Yaskawa INFORM job: u_tourne2TRJ2.JBI

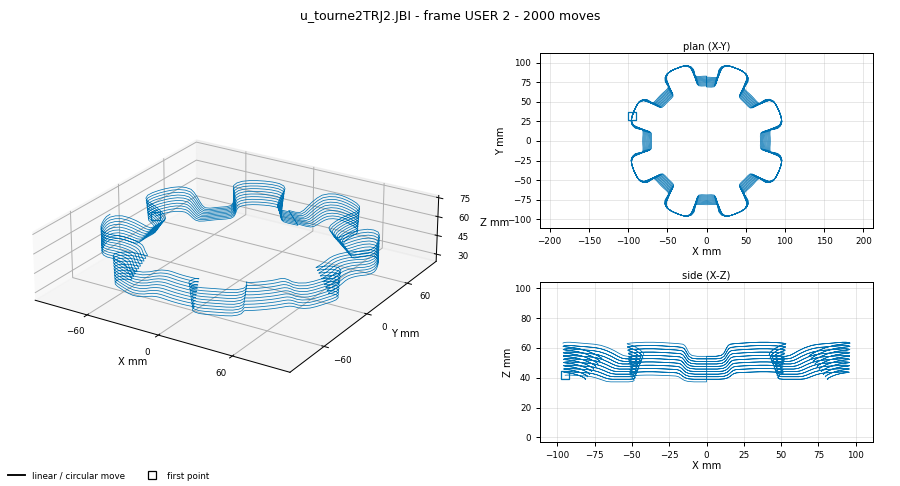
[picture p0: tool path of u_tourne2TRJ2.JBI in frame USER 2, 2000 of 2000 moves have a stored position in this frame; points joined in program order, loops and branches not executed]
/JOB
//NAME u_tourne2TRJ2
///FOLDERNAME DEMO
//POS
///NPOS 2000,0,0,0,0,0
///USER 2
///TOOL 7
///POSTYPE USER
///RECTAN
///RCONF 1,0,0,0,0,0,0,0,0,0,0,0,0,0,0,0,0,0,0,0,0,0,0,0
C00000=-94.679,31.992,41.678,179.9828,-0.0630,0.0000
C00001=-93.214,36.189,41.785,179.9943,-0.0057,0.0000
C00002=-91.502,40.323,41.785,179.9943,-0.0057,0.0000
C00003=-89.570,44.326,41.678,179.9714,-0.0573,0.0000
C00004=-87.153,47.905,41.515,178.9971,-1.0602,0.0000
C00005=-83.964,50.341,41.355,177.9939,-1.0435,0.0000
C00006=-80.606,51.270,41.159,176.0662,-0.0632,0.0000
C00007=-77.545,50.645,40.789,176.2839,1.1369,0.0000
C00008=-74.511,49.565,40.048,179.1806,0.2980,0.0000
C00009=-71.724,48.673,39.090,-174.7314,-1.4558,0.0000
C00010=-69.261,48.447,38.165,-161.9039,-0.3255,0.0000
C00011=-66.868,49.465,37.495,-150.1012,20.4852,0.0000
C00012=-64.059,52.288,37.229,-152.5935,29.6888,0.0000
C00013=-61.349,55.398,37.217,-152.6199,30.0128,0.0000
C00014=-58.451,58.451,37.225,-151.2622,28.7378,0.0000
C00015=-55.398,61.349,37.217,-149.9872,27.3801,0.0000
C00016=-52.288,64.059,37.229,-150.3112,27.4065,0.0000
C00017=-49.465,66.868,37.495,-159.5087,29.8988,0.0000
C00018=-48.447,69.261,38.165,179.6745,18.0961,0.0000
C00019=-48.673,71.724,39.090,178.5442,5.2686,0.0000
C00020=-49.565,74.511,40.048,-179.7020,-0.8194,0.0000
C00021=-50.645,77.545,40.789,-178.8631,-3.7161,0.0000
C00022=-51.270,80.606,41.159,179.9368,-3.9338,0.0000
C00023=-50.341,83.964,41.355,178.9565,-2.0061,0.0000
C00024=-47.905,87.153,41.515,178.9398,-1.0029,0.0000
C00025=-44.326,89.570,41.678,179.9427,-0.0286,0.0000
C00026=-40.323,91.502,41.785,179.9943,-0.0057,0.0000
C00027=-36.189,93.214,41.785,179.9943,-0.0057,0.0000
C00028=-31.992,94.679,41.678,179.9370,-0.0172,0.0000
C00029=-27.752,95.500,41.515,178.5446,-0.0401,0.0000
C00030=-23.775,94.968,41.355,177.8450,0.6823,0.0000
C00031=-20.743,93.250,41.159,177.1708,2.7375,0.0000
C00032=-19.021,90.644,40.789,178.1744,3.4301,0.0000
C00033=-17.640,87.735,40.048,179.6333,0.7850,0.0000
C00034=-16.299,85.134,39.090,-177.2969,-4.7546,0.0000
C00035=-14.718,83.232,38.165,-167.2085,-13.2264,0.0000
C00036=-12.305,82.260,37.495,-146.1467,-8.1019,0.0000
C00037=-8.324,82.270,37.229,-142.4136,2.0895,0.0000
C00038=-4.208,82.553,37.217,-142.2346,2.4206,0.0000
C00039=0.000,82.662,37.225,-142.2064,0.0000,0.0000
C00040=0.000,81.307,38.958,-141.7572,0.0000,0.0000
C00041=4.084,81.202,38.949,-141.7896,-2.4427,0.0000
C00042=8.115,80.931,38.962,-141.9757,-1.8546,0.0000
C00043=12.050,80.963,39.253,-146.2971,9.3078,0.0000
C00044=14.402,82.041,39.987,-169.0733,12.6730,0.0000
C00045=15.932,84.113,41.004,-178.0935,3.7115,0.0000
C00046=17.234,86.943,42.060,179.2949,-1.6619,0.0000
C00047=18.580,90.119,42.880,177.9599,-4.2637,0.0000
C00048=20.259,92.987,43.289,176.7667,-3.4911,0.0000
C00049=23.317,94.913,43.506,177.4435,-0.9062,0.0000
C00050=27.389,95.566,43.684,178.3669,0.0229,0.0000
C00051=31.762,94.755,43.864,179.9255,0.0229,0.0000
C00052=36.110,93.244,43.984,179.9885,0.0057,0.0000
C00053=40.400,91.468,43.984,179.9885,0.0057,0.0000
C00054=44.543,89.461,43.864,179.9312,0.0344,0.0000
C00055=48.209,86.942,43.684,178.8309,1.1405,0.0000
C00056=50.626,83.601,43.506,178.8358,2.4477,0.0000
C00057=51.426,80.077,43.289,-179.8160,4.7437,0.0000
C00058=50.586,76.861,42.880,-178.4251,4.4523,0.0000
C00059=49.291,73.664,42.060,-179.3236,1.6734,0.0000
C00060=48.211,70.742,41.004,178.7192,-3.9688,0.0000
C00061=47.828,68.195,39.987,178.7094,-16.4610,0.0000
C00062=48.729,65.770,39.253,-160.4136,-30.4355,0.0000
C00063=51.488,62.965,38.962,-150.0635,-27.9250,0.0000
C00064=54.531,60.307,38.949,-149.5964,-27.7691,0.0000
C00065=57.493,57.493,38.958,-150.8693,-29.1307,0.0000
C00066=60.306,54.531,38.949,-152.2309,-30.4036,0.0000
C00067=62.965,51.488,38.962,-152.0750,-29.9365,0.0000
C00068=65.770,48.729,39.253,-149.5645,-19.5864,0.0000
C00069=68.195,47.828,39.987,-163.5390,1.2906,0.0000
C00070=70.742,48.211,41.004,-176.0312,1.2808,0.0000
C00071=73.664,49.291,42.060,178.3266,-0.6764,0.0000
C00072=76.861,50.586,42.880,175.5477,-1.5749,0.0000
C00073=80.077,51.426,43.289,175.2563,-0.1840,0.0000
C00074=83.601,50.626,43.506,177.5523,1.1642,0.0000
C00075=86.942,48.209,43.684,178.8595,1.1691,0.0000
C00076=89.461,44.543,43.864,179.9656,0.0688,0.0000
C00077=91.468,40.400,43.984,179.9943,0.0115,0.0000
C00078=93.244,36.110,43.984,179.9943,0.0115,0.0000
C00079=94.755,31.762,43.864,179.9771,0.0745,0.0000
C00080=95.566,27.389,43.684,179.9771,1.6331,0.0000
C00081=94.913,23.317,43.506,-179.0938,2.5565,0.0000
C00082=92.987,20.259,43.289,-176.5089,3.2333,0.0000
C00083=90.119,18.580,42.880,-175.7363,2.0401,0.0000
C00084=86.943,17.234,42.060,-178.3381,0.7051,0.0000
C00085=84.113,15.932,41.004,176.2885,-1.9065,0.0000
C00086=82.041,14.402,39.987,167.3270,-10.9267,0.0000
C00087=80.963,12.050,39.253,170.6922,-33.7029,0.0000
C00088=80.931,8.115,38.962,-178.1454,-38.0243,0.0000
C00089=81.202,4.084,38.949,-177.5573,-38.2104,0.0000
C00090=81.307,0.000,38.958,180.0000,-38.2428,0.0000
C00091=81.202,-4.084,38.949,177.5573,-38.2104,0.0000
C00092=80.931,-8.116,38.962,178.1454,-38.0243,0.0000
C00093=80.963,-12.050,39.253,-170.6922,-33.7029,0.0000
C00094=82.041,-14.402,39.987,-167.3270,-10.9267,0.0000
C00095=84.113,-15.932,41.004,-176.2885,-1.9065,0.0000
C00096=86.943,-17.234,42.060,178.3381,0.7051,0.0000
C00097=90.119,-18.580,42.880,175.7363,2.0401,0.0000
C00098=92.987,-20.259,43.289,176.5089,3.2333,0.0000
C00099=94.913,-23.317,43.506,179.0938,2.5565,0.0000
C00100=95.566,-27.389,43.684,-179.9771,1.6331,0.0000
C00101=94.755,-31.762,43.864,-179.9771,0.0745,0.0000
C00102=93.244,-36.110,43.984,-179.9943,0.0115,0.0000
C00103=91.468,-40.400,43.984,-179.9943,0.0115,0.0000
C00104=89.461,-44.543,43.864,-179.9656,0.0688,0.0000
C00105=86.942,-48.209,43.684,-178.8595,1.1691,0.0000
C00106=83.601,-50.626,43.506,-177.5523,1.1642,0.0000
C00107=80.077,-51.426,43.289,-175.2563,-0.1840,0.0000
C00108=76.861,-50.586,42.880,-175.5477,-1.5749,0.0000
C00109=73.664,-49.291,42.060,-178.3266,-0.6764,0.0000
C00110=70.742,-48.211,41.004,176.0312,1.2808,0.0000
C00111=68.195,-47.828,39.987,163.5390,1.2906,0.0000
C00112=65.770,-48.729,39.253,149.5645,-19.5864,0.0000
C00113=62.965,-51.488,38.962,152.0750,-29.9365,0.0000
C00114=60.307,-54.531,38.949,152.2309,-30.4036,0.0000
C00115=57.493,-57.493,38.958,150.8693,-29.1307,0.0000
C00116=54.531,-60.306,38.949,149.5964,-27.7691,0.0000
C00117=51.488,-62.965,38.962,150.0635,-27.9250,0.0000
C00118=48.729,-65.770,39.253,160.4136,-30.4355,0.0000
C00119=47.828,-68.195,39.987,-178.7094,-16.4610,0.0000
C00120=48.211,-70.742,41.004,-178.7192,-3.9688,0.0000
C00121=49.291,-73.664,42.060,179.3236,1.6734,0.0000
C00122=50.586,-76.861,42.880,178.4251,4.4523,0.0000
C00123=51.426,-80.077,43.289,179.8160,4.7437,0.0000
C00124=50.626,-83.601,43.506,-178.8358,2.4477,0.0000
C00125=48.209,-86.942,43.684,-178.8309,1.1405,0.0000
C00126=44.543,-89.461,43.864,-179.9312,0.0344,0.0000
C00127=40.400,-91.468,43.984,-179.9885,0.0057,0.0000
C00128=36.110,-93.244,43.984,-179.9885,0.0057,0.0000
C00129=31.762,-94.755,43.864,-179.9255,0.0229,0.0000
C00130=27.389,-95.566,43.684,-178.3669,0.0229,0.0000
C00131=23.317,-94.913,43.506,-177.4435,-0.9062,0.0000
C00132=20.259,-92.987,43.289,-176.7667,-3.4911,0.0000
C00133=18.580,-90.119,42.880,-177.9599,-4.2637,0.0000
C00134=17.234,-86.943,42.060,-179.2949,-1.6619,0.0000
C00135=15.932,-84.113,41.004,178.0935,3.7115,0.0000
C00136=14.402,-82.041,39.987,169.0733,12.6730,0.0000
C00137=12.050,-80.963,39.253,146.2971,9.3078,0.0000
C00138=8.115,-80.931,38.962,141.9757,-1.8546,0.0000
C00139=4.084,-81.202,38.949,141.7896,-2.4427,0.0000
C00140=0.000,-81.307,38.958,141.7572,0.0000,0.0000
C00141=0.000,-81.307,38.958,141.7572,0.0000,0.0000
C00142=-4.084,-81.202,38.949,141.7896,2.4427,0.0000
C00143=-8.116,-80.931,38.962,141.9757,1.8546,0.0000
C00144=-12.050,-80.963,39.253,146.2971,-9.3078,0.0000
C00145=-14.402,-82.041,39.987,169.0733,-12.6730,0.0000
C00146=-15.932,-84.113,41.004,178.0935,-3.7115,0.0000
C00147=-17.234,-86.943,42.060,-179.2949,1.6619,0.0000
C00148=-18.580,-90.119,42.880,-177.9599,4.2637,0.0000
C00149=-20.259,-92.987,43.289,-176.7667,3.4911,0.0000
C00150=-23.317,-94.913,43.506,-177.4435,0.9062,0.0000
C00151=-27.389,-95.566,43.684,-178.3669,-0.0229,0.0000
C00152=-31.762,-94.755,43.864,-179.9255,-0.0229,0.0000
C00153=-36.110,-93.244,43.984,-179.9885,-0.0057,0.0000
C00154=-40.400,-91.468,43.984,-179.9885,-0.0057,0.0000
C00155=-44.543,-89.461,43.864,-179.9312,-0.0344,0.0000
C00156=-48.209,-86.942,43.684,-178.8309,-1.1405,0.0000
C00157=-50.626,-83.601,43.506,-178.8358,-2.4477,0.0000
C00158=-51.426,-80.077,43.289,179.8160,-4.7437,0.0000
C00159=-50.586,-76.861,42.880,178.4251,-4.4523,0.0000
C00160=-49.291,-73.664,42.060,179.3236,-1.6734,0.0000
C00161=-48.211,-70.742,41.004,-178.7192,3.9688,0.0000
C00162=-47.828,-68.195,39.987,-178.7094,16.4610,0.0000
C00163=-48.729,-65.770,39.253,160.4136,30.4355,0.0000
C00164=-51.488,-62.965,38.962,150.0635,27.9250,0.0000
C00165=-54.531,-60.307,38.949,149.5964,27.7691,0.0000
C00166=-57.493,-57.493,38.958,150.8693,29.1307,0.0000
C00167=-60.306,-54.531,38.949,152.2309,30.4036,0.0000
C00168=-62.965,-51.488,38.962,152.0750,29.9365,0.0000
C00169=-65.770,-48.729,39.253,149.5645,19.5864,0.0000
C00170=-68.195,-47.828,39.987,163.5390,-1.2906,0.0000
C00171=-70.742,-48.211,41.004,176.0312,-1.2808,0.0000
C00172=-73.664,-49.291,42.060,-178.3266,0.6764,0.0000
C00173=-76.861,-50.586,42.880,-175.5477,1.5749,0.0000
C00174=-80.077,-51.426,43.289,-175.2563,0.1840,0.0000
C00175=-83.601,-50.626,43.506,-177.5523,-1.1642,0.0000
C00176=-86.942,-48.209,43.684,-178.8595,-1.1691,0.0000
C00177=-89.461,-44.543,43.864,-179.9656,-0.0688,0.0000
C00178=-91.468,-40.400,43.984,-179.9943,-0.0115,0.0000
C00179=-93.244,-36.110,43.984,-179.9943,-0.0115,0.0000
C00180=-94.755,-31.762,43.864,-179.9771,-0.0745,0.0000
C00181=-95.566,-27.389,43.684,-179.9771,-1.6331,0.0000
C00182=-94.913,-23.317,43.506,179.0938,-2.5565,0.0000
C00183=-92.987,-20.259,43.289,176.5089,-3.2333,0.0000
C00184=-90.119,-18.580,42.880,175.7363,-2.0401,0.0000
C00185=-86.943,-17.234,42.060,178.3381,-0.7051,0.0000
C00186=-84.113,-15.932,41.004,-176.2885,1.9065,0.0000
C00187=-82.041,-14.402,39.987,-167.3270,10.9267,0.0000
C00188=-80.963,-12.050,39.253,-170.6922,33.7029,0.0000
C00189=-80.931,-8.115,38.962,178.1454,38.0243,0.0000
C00190=-81.202,-4.084,38.949,177.5573,38.2104,0.0000
C00191=-81.307,0.000,38.958,-180.0000,38.2428,0.0000
C00192=-81.202,4.084,38.949,-177.5573,38.2104,0.0000
C00193=-80.931,8.116,38.962,-178.1454,38.0243,0.0000
C00194=-80.963,12.050,39.253,170.6922,33.7029,0.0000
C00195=-82.041,14.402,39.987,167.3270,10.9267,0.0000
C00196=-84.113,15.932,41.004,176.2885,1.9065,0.0000
C00197=-86.943,17.234,42.060,-178.3381,-0.7051,0.0000
C00198=-90.119,18.580,42.880,-175.7363,-2.0401,0.0000
C00199=-92.987,20.259,43.289,-176.5089,-3.2333,0.0000
C00200=-94.913,23.317,43.506,-179.0938,-2.5565,0.0000
C00201=-95.566,27.389,43.684,179.9771,-1.6331,0.0000
C00202=-94.755,31.762,43.864,179.9771,-0.0745,0.0000
C00203=-93.244,36.110,43.984,179.9943,-0.0115,0.0000
C00204=-91.468,40.400,43.984,179.9943,-0.0115,0.0000
C00205=-89.461,44.543,43.864,179.9656,-0.0688,0.0000
C00206=-86.942,48.209,43.684,178.8595,-1.1691,0.0000
C00207=-83.601,50.626,43.506,177.5523,-1.1642,0.0000
C00208=-80.077,51.426,43.289,175.2563,0.1840,0.0000
C00209=-76.861,50.586,42.880,175.5477,1.5749,0.0000
C00210=-73.664,49.291,42.060,178.3266,0.6764,0.0000
C00211=-70.742,48.211,41.004,-176.0312,-1.2808,0.0000
C00212=-68.195,47.828,39.987,-163.5390,-1.2906,0.0000
C00213=-65.770,48.729,39.253,-149.5645,19.5864,0.0000
C00214=-62.965,51.488,38.962,-152.0750,29.9365,0.0000
C00215=-60.307,54.531,38.949,-152.2309,30.4036,0.0000
C00216=-57.493,57.493,38.958,-150.8693,29.1307,0.0000
C00217=-54.531,60.306,38.949,-149.5964,27.7691,0.0000
C00218=-51.488,62.965,38.962,-150.0635,27.9250,0.0000
C00219=-48.729,65.770,39.253,-160.4136,30.4355,0.0000
C00220=-47.828,68.195,39.987,178.7094,16.4610,0.0000
C00221=-48.211,70.742,41.004,178.7192,3.9688,0.0000
C00222=-49.291,73.664,42.060,-179.3236,-1.6734,0.0000
C00223=-50.586,76.861,42.880,-178.4251,-4.4523,0.0000
C00224=-51.426,80.077,43.289,-179.8160,-4.7437,0.0000
C00225=-50.626,83.601,43.506,178.8358,-2.4477,0.0000
C00226=-48.209,86.942,43.684,178.8309,-1.1405,0.0000
C00227=-44.543,89.461,43.864,179.9312,-0.0344,0.0000
C00228=-40.400,91.468,43.984,179.9885,-0.0057,0.0000
C00229=-36.110,93.244,43.984,179.9885,-0.0057,0.0000
C00230=-31.762,94.755,43.864,179.9255,-0.0229,0.0000
C00231=-27.389,95.566,43.684,178.3669,-0.0229,0.0000
C00232=-23.317,94.913,43.506,177.4435,0.9062,0.0000
C00233=-20.259,92.987,43.289,176.7667,3.4911,0.0000
C00234=-18.580,90.119,42.880,177.9599,4.2637,0.0000
C00235=-17.234,86.943,42.060,179.2949,1.6619,0.0000
C00236=-15.932,84.113,41.004,-178.0935,-3.7115,0.0000
C00237=-14.402,82.041,39.987,-169.0733,-12.6730,0.0000
C00238=-12.050,80.963,39.253,-146.2971,-9.3078,0.0000
C00239=-8.116,80.931,38.962,-141.9757,1.8546,0.0000
C00240=-4.084,81.202,38.949,-141.7896,2.4427,0.0000
C00241=0.000,81.307,38.958,-141.7572,0.0000,0.0000
C00242=0.000,79.940,40.681,-141.3939,0.0000,0.0000
C00243=3.959,79.840,40.672,-141.4226,-2.4552,0.0000
C00244=7.905,79.580,40.686,-141.6239,-1.6005,0.0000
C00245=11.791,79.654,41.003,-146.5977,10.4649,0.0000
C00246=14.083,80.839,41.802,-170.8080,11.8958,0.0000
C00247=15.561,83.082,42.912,-178.7438,2.7001,0.0000
C00248=16.825,86.143,44.068,179.0422,-2.4592,0.0000
C00249=18.134,89.588,44.968,177.8312,-5.0060,0.0000
C00250=19.771,92.721,45.418,176.4760,-4.2001,0.0000
C00251=22.856,94.857,45.657,177.0818,-1.1475,0.0000
C00252=27.022,95.633,45.852,178.2006,-0.0057,0.0000
C00253=31.529,94.831,46.051,179.9083,0.0286,0.0000
C00254=36.031,93.275,46.182,179.9885,0.0057,0.0000
C00255=40.478,91.433,46.182,179.9885,0.0057,0.0000
C00256=44.762,89.350,46.051,179.9141,0.0458,0.0000
C00257=48.515,86.730,45.852,178.7333,1.2781,0.0000
C00258=50.913,83.236,45.657,178.7493,2.8724,0.0000
C00259=51.583,79.544,45.418,-179.5165,5.4517,0.0000
C00260=50.526,76.172,44.968,-177.9864,5.0688,0.0000
C00261=49.015,72.810,44.068,-178.9332,2.4134,0.0000
C00262=47.744,69.752,42.912,178.9789,-2.7974,0.0000
C00263=47.203,67.120,41.802,178.0208,-14.7523,0.0000
C00264=47.986,64.662,41.003,-161.4422,-30.8329,0.0000
C00265=50.682,61.862,40.686,-149.9029,-28.3774,0.0000
C00266=53.655,59.255,40.672,-149.2730,-28.0900,0.0000
C00267=56.526,56.526,40.681,-150.5529,-29.4471,0.0000
C00268=59.255,53.656,40.672,-151.9100,-30.7270,0.0000
C00269=61.862,50.682,40.686,-151.6226,-30.0971,0.0000
C00270=64.662,47.986,41.003,-149.1671,-18.5578,0.0000
C00271=67.120,47.203,41.802,-165.2477,1.9792,0.0000
C00272=69.752,47.744,42.912,-177.2026,1.0211,0.0000
C00273=72.810,49.015,44.068,177.5866,-1.0668,0.0000
C00274=76.172,50.526,44.968,174.9312,-2.0136,0.0000
C00275=79.544,51.583,45.418,174.5483,-0.4835,0.0000
C00276=83.236,50.913,45.657,177.1276,1.2507,0.0000
C00277=86.730,48.515,45.852,178.7219,1.2667,0.0000
C00278=89.350,44.762,46.051,179.9542,0.0859,0.0000
C00279=91.433,40.478,46.182,179.9943,0.0115,0.0000
C00280=93.275,36.031,46.182,179.9943,0.0115,0.0000
C00281=94.831,31.529,46.051,179.9714,0.0917,0.0000
C00282=95.633,27.022,45.852,-179.9943,1.7994,0.0000
C00283=94.857,22.856,45.657,-178.8525,2.9182,0.0000
C00284=92.721,19.771,45.418,-175.7999,3.5240,0.0000
C00285=89.588,18.134,44.968,-174.9940,2.1688,0.0000
C00286=86.143,16.825,44.068,-177.5408,0.9578,0.0000
C00287=83.082,15.561,42.912,177.2999,-1.2562,0.0000
C00288=80.839,14.083,41.802,168.1042,-9.1920,0.0000
C00289=79.654,11.791,41.003,169.5351,-33.4023,0.0000
C00290=79.580,7.905,40.686,-178.3995,-38.3761,0.0000
C00291=79.840,3.959,40.672,-177.5448,-38.5774,0.0000
C00292=79.940,0.000,40.681,180.0000,-38.6061,0.0000
C00293=79.840,-3.959,40.672,177.5448,-38.5774,0.0000
C00294=79.580,-7.905,40.686,178.3995,-38.3716,0.0000
C00295=79.654,-11.792,41.003,-169.5351,-33.4023,0.0000
C00296=80.839,-14.083,41.802,-168.1042,-9.1920,0.0000
C00297=83.082,-15.561,42.912,-177.2999,-1.2562,0.0000
C00298=86.143,-16.825,44.068,177.5408,0.9578,0.0000
C00299=89.588,-18.134,44.968,174.9940,2.1688,0.0000
C00300=92.721,-19.771,45.418,175.7999,3.5240,0.0000
C00301=94.857,-22.856,45.657,178.8525,2.9182,0.0000
C00302=95.633,-27.022,45.852,179.9943,1.7994,0.0000
C00303=94.831,-31.529,46.051,-179.9714,0.0917,0.0000
C00304=93.275,-36.031,46.182,-179.9943,0.0115,0.0000
C00305=91.433,-40.478,46.182,-179.9943,0.0115,0.0000
C00306=89.350,-44.762,46.051,-179.9542,0.0859,0.0000
C00307=86.730,-48.515,45.852,-178.7219,1.2667,0.0000
C00308=83.236,-50.913,45.657,-177.1276,1.2507,0.0000
C00309=79.544,-51.583,45.418,-174.5483,-0.4835,0.0000
C00310=76.172,-50.526,44.968,-174.9312,-2.0136,0.0000
C00311=72.810,-49.015,44.068,-177.5866,-1.0668,0.0000
C00312=69.752,-47.744,42.912,177.2026,1.0211,0.0000
C00313=67.120,-47.203,41.802,165.2477,1.9792,0.0000
C00314=64.662,-47.986,41.003,149.1671,-18.5578,0.0000
C00315=61.862,-50.682,40.686,151.6226,-30.0971,0.0000
C00316=59.255,-53.655,40.672,151.9100,-30.7270,0.0000
C00317=56.526,-56.526,40.681,150.5529,-29.4471,0.0000
C00318=53.656,-59.255,40.672,149.2730,-28.0900,0.0000
C00319=50.682,-61.862,40.686,149.9029,-28.3774,0.0000
C00320=47.986,-64.662,41.003,161.4422,-30.8329,0.0000
C00321=47.203,-67.120,41.802,-178.0208,-14.7523,0.0000
C00322=47.744,-69.752,42.912,-178.9789,-2.7974,0.0000
C00323=49.015,-72.810,44.068,178.9332,2.4134,0.0000
C00324=50.526,-76.172,44.968,177.9864,5.0688,0.0000
C00325=51.583,-79.544,45.418,179.5165,5.4517,0.0000
C00326=50.913,-83.236,45.657,-178.7493,2.8724,0.0000
C00327=48.515,-86.730,45.852,-178.7333,1.2781,0.0000
C00328=44.762,-89.350,46.051,-179.9141,0.0458,0.0000
C00329=40.478,-91.433,46.182,-179.9885,0.0057,0.0000
C00330=36.031,-93.275,46.182,-179.9885,0.0057,0.0000
C00331=31.529,-94.831,46.051,-179.9083,0.0286,0.0000
C00332=27.022,-95.633,45.852,-178.2006,-0.0057,0.0000
C00333=22.856,-94.857,45.657,-177.0818,-1.1475,0.0000
C00334=19.771,-92.721,45.418,-176.4760,-4.2001,0.0000
C00335=18.134,-89.588,44.968,-177.8312,-5.0060,0.0000
C00336=16.825,-86.143,44.068,-179.0422,-2.4592,0.0000
C00337=15.561,-83.082,42.912,178.7438,2.7001,0.0000
C00338=14.083,-80.839,41.802,170.8080,11.8958,0.0000
C00339=11.791,-79.654,41.003,146.5977,10.4649,0.0000
C00340=7.905,-79.580,40.686,141.6239,-1.6005,0.0000
C00341=3.959,-79.840,40.672,141.4226,-2.4552,0.0000
C00342=0.000,-79.940,40.681,141.3939,0.0000,0.0000
C00343=0.000,-79.940,40.681,141.3939,0.0000,0.0000
C00344=-3.959,-79.840,40.672,141.4226,2.4552,0.0000
C00345=-7.905,-79.580,40.686,141.6284,1.6005,0.0000
C00346=-11.792,-79.654,41.003,146.5977,-10.4649,0.0000
C00347=-14.083,-80.839,41.802,170.8080,-11.8958,0.0000
C00348=-15.561,-83.082,42.912,178.7438,-2.7001,0.0000
C00349=-16.825,-86.143,44.068,-179.0422,2.4592,0.0000
C00350=-18.134,-89.588,44.968,-177.8312,5.0060,0.0000
C00351=-19.771,-92.721,45.418,-176.4760,4.2001,0.0000
C00352=-22.856,-94.857,45.657,-177.0818,1.1475,0.0000
C00353=-27.022,-95.633,45.852,-178.2006,0.0057,0.0000
C00354=-31.529,-94.831,46.051,-179.9083,-0.0286,0.0000
C00355=-36.031,-93.275,46.182,-179.9885,-0.0057,0.0000
C00356=-40.478,-91.433,46.182,-179.9885,-0.0057,0.0000
C00357=-44.762,-89.350,46.051,-179.9141,-0.0458,0.0000
C00358=-48.515,-86.730,45.852,-178.7333,-1.2781,0.0000
C00359=-50.913,-83.236,45.657,-178.7493,-2.8724,0.0000
C00360=-51.583,-79.544,45.418,179.5165,-5.4517,0.0000
C00361=-50.526,-76.172,44.968,177.9864,-5.0688,0.0000
C00362=-49.015,-72.810,44.068,178.9332,-2.4134,0.0000
C00363=-47.744,-69.752,42.912,-178.9789,2.7974,0.0000
C00364=-47.203,-67.120,41.802,-178.0208,14.7523,0.0000
C00365=-47.986,-64.662,41.003,161.4422,30.8329,0.0000
C00366=-50.682,-61.862,40.686,149.9029,28.3774,0.0000
C00367=-53.655,-59.255,40.672,149.2730,28.0900,0.0000
C00368=-56.526,-56.526,40.681,150.5529,29.4471,0.0000
C00369=-59.255,-53.656,40.672,151.9100,30.7270,0.0000
C00370=-61.862,-50.682,40.686,151.6226,30.0971,0.0000
C00371=-64.662,-47.986,41.003,149.1671,18.5578,0.0000
C00372=-67.120,-47.203,41.802,165.2477,-1.9792,0.0000
C00373=-69.752,-47.744,42.912,177.2026,-1.0211,0.0000
C00374=-72.810,-49.015,44.068,-177.5866,1.0668,0.0000
C00375=-76.172,-50.526,44.968,-174.9312,2.0136,0.0000
C00376=-79.544,-51.583,45.418,-174.5483,0.4835,0.0000
C00377=-83.236,-50.913,45.657,-177.1276,-1.2507,0.0000
C00378=-86.730,-48.515,45.852,-178.7219,-1.2667,0.0000
C00379=-89.350,-44.762,46.051,-179.9542,-0.0859,0.0000
C00380=-91.433,-40.478,46.182,-179.9943,-0.0115,0.0000
C00381=-93.275,-36.031,46.182,-179.9943,-0.0115,0.0000
C00382=-94.831,-31.529,46.051,-179.9714,-0.0917,0.0000
C00383=-95.633,-27.022,45.852,179.9943,-1.7994,0.0000
C00384=-94.857,-22.856,45.657,178.8525,-2.9182,0.0000
C00385=-92.721,-19.771,45.418,175.7999,-3.5240,0.0000
C00386=-89.588,-18.134,44.968,174.9940,-2.1688,0.0000
C00387=-86.143,-16.825,44.068,177.5408,-0.9578,0.0000
C00388=-83.082,-15.561,42.912,-177.2999,1.2562,0.0000
C00389=-80.839,-14.083,41.802,-168.1042,9.1920,0.0000
C00390=-79.654,-11.791,41.003,-169.5351,33.4023,0.0000
C00391=-79.580,-7.905,40.686,178.3995,38.3761,0.0000
C00392=-79.840,-3.959,40.672,177.5448,38.5774,0.0000
C00393=-79.940,0.000,40.681,-180.0000,38.6061,0.0000
C00394=-79.840,3.959,40.672,-177.5448,38.5774,0.0000
C00395=-79.580,7.905,40.686,-178.3995,38.3716,0.0000
C00396=-79.654,11.792,41.003,169.5351,33.4023,0.0000
C00397=-80.839,14.083,41.802,168.1042,9.1920,0.0000
C00398=-83.082,15.561,42.912,177.2999,1.2562,0.0000
C00399=-86.143,16.825,44.068,-177.5408,-0.9578,0.0000
C00400=-89.588,18.134,44.968,-174.9940,-2.1688,0.0000
C00401=-92.721,19.771,45.418,-175.7999,-3.5240,0.0000
C00402=-94.857,22.856,45.657,-178.8525,-2.9182,0.0000
C00403=-95.633,27.022,45.852,-179.9943,-1.7994,0.0000
C00404=-94.831,31.529,46.051,179.9714,-0.0917,0.0000
C00405=-93.275,36.031,46.182,179.9943,-0.0115,0.0000
C00406=-91.433,40.478,46.182,179.9943,-0.0115,0.0000
C00407=-89.350,44.762,46.051,179.9542,-0.0859,0.0000
C00408=-86.730,48.515,45.852,178.7219,-1.2667,0.0000
C00409=-83.236,50.913,45.657,177.1276,-1.2507,0.0000
C00410=-79.544,51.583,45.418,174.5483,0.4835,0.0000
C00411=-76.172,50.526,44.968,174.9312,2.0136,0.0000
C00412=-72.810,49.015,44.068,177.5866,1.0668,0.0000
C00413=-69.752,47.744,42.912,-177.2026,-1.0211,0.0000
C00414=-67.120,47.203,41.802,-165.2477,-1.9792,0.0000
C00415=-64.662,47.986,41.003,-149.1671,18.5578,0.0000
C00416=-61.862,50.682,40.686,-151.6226,30.0971,0.0000
C00417=-59.255,53.655,40.672,-151.9100,30.7270,0.0000
C00418=-56.526,56.526,40.681,-150.5529,29.4471,0.0000
C00419=-53.656,59.255,40.672,-149.2730,28.0900,0.0000
C00420=-50.682,61.862,40.686,-149.9029,28.3774,0.0000
C00421=-47.986,64.662,41.003,-161.4422,30.8329,0.0000
C00422=-47.203,67.120,41.802,178.0208,14.7523,0.0000
C00423=-47.744,69.752,42.912,178.9789,2.7974,0.0000
C00424=-49.015,72.810,44.068,-178.9332,-2.4134,0.0000
C00425=-50.526,76.172,44.968,-177.9864,-5.0688,0.0000
C00426=-51.583,79.544,45.418,-179.5165,-5.4517,0.0000
C00427=-50.913,83.236,45.657,178.7493,-2.8724,0.0000
C00428=-48.515,86.730,45.852,178.7333,-1.2781,0.0000
C00429=-44.762,89.350,46.051,179.9141,-0.0458,0.0000
C00430=-40.478,91.433,46.182,179.9885,-0.0057,0.0000
C00431=-36.031,93.275,46.182,179.9885,-0.0057,0.0000
C00432=-31.529,94.831,46.051,179.9083,-0.0286,0.0000
C00433=-27.022,95.633,45.852,178.2006,0.0057,0.0000
C00434=-22.856,94.857,45.657,177.0818,1.1475,0.0000
C00435=-19.771,92.721,45.418,176.4760,4.2001,0.0000
C00436=-18.134,89.588,44.968,177.8312,5.0060,0.0000
C00437=-16.825,86.143,44.068,179.0422,2.4592,0.0000
C00438=-15.561,83.082,42.912,-178.7438,-2.7001,0.0000
C00439=-14.083,80.839,41.802,-170.8080,-11.8958,0.0000
C00440=-11.792,79.654,41.003,-146.5977,-10.4649,0.0000
C00441=-7.905,79.580,40.686,-141.6284,1.6005,0.0000
C00442=-3.959,79.840,40.672,-141.4226,2.4552,0.0000
C00443=0.000,79.940,40.681,-141.3939,0.0000,0.0000
C00444=0.000,78.562,42.397,-141.1129,0.0000,0.0000
C00445=3.833,78.467,42.387,-141.1370,-2.4576,0.0000
C00446=7.694,78.220,42.402,-141.3590,-1.3205,0.0000
C00447=11.532,78.336,42.745,-147.0419,11.5629,0.0000
C00448=13.762,79.628,43.611,-172.3757,10.9597,0.0000
C00449=15.189,82.045,44.816,-179.2606,1.7364,0.0000
C00450=16.414,85.339,46.074,178.8695,-3.1763,0.0000
C00451=17.687,89.056,47.055,177.7713,-5.6570,0.0000
C00452=19.281,92.454,47.546,176.2827,-4.8633,0.0000
C00453=22.392,94.802,47.807,176.7658,-1.3947,0.0000
C00454=26.654,95.700,48.020,178.0515,-0.0344,0.0000
C00455=31.296,94.909,48.237,179.8969,0.0344,0.0000
C00456=35.952,93.306,48.381,179.9885,0.0057,0.0000
C00457=40.555,91.399,48.381,179.9885,0.0057,0.0000
C00458=44.981,89.240,48.237,179.9026,0.0516,0.0000
C00459=48.823,86.517,48.020,178.6473,1.4043,0.0000
C00460=51.201,82.869,47.807,178.6971,3.2685,0.0000
C00461=51.741,79.009,47.546,-179.1876,6.0567,0.0000
C00462=50.465,75.478,47.055,-177.5642,5.5714,0.0000
C00463=48.737,71.950,46.074,-178.5540,3.0447,0.0000
C00464=47.275,68.755,44.816,179.2949,-1.7479,0.0000
C00465=46.575,66.037,43.611,177.5764,-13.0376,0.0000
C00466=47.238,63.546,42.745,-162.5789,-31.0909,0.0000
C00467=49.870,60.750,42.402,-149.8162,-28.7716,0.0000
C00468=52.774,58.195,42.387,-149.0319,-28.3446,0.0000
C00469=55.552,55.552,42.397,-150.3051,-29.6949,0.0000
C00470=58.195,52.774,42.387,-151.6554,-30.9681,0.0000
C00471=60.750,49.870,42.402,-151.2315,-30.1807,0.0000
C00472=63.546,47.238,42.745,-148.9091,-17.4211,0.0000
C00473=66.037,46.575,43.611,-166.9624,2.4236,0.0000
C00474=68.755,47.275,44.816,-178.2521,0.7051,0.0000
C00475=71.950,48.737,46.074,176.9553,-1.4460,0.0000
C00476=75.478,50.465,47.055,174.4286,-2.4358,0.0000
C00477=79.009,51.741,47.546,173.9433,-0.8124,0.0000
C00478=82.869,51.201,47.807,176.7315,1.3029,0.0000
C00479=86.517,48.823,48.020,178.5957,1.3527,0.0000
C00480=89.240,44.981,48.237,179.9484,0.0974,0.0000
C00481=91.399,40.555,48.381,179.9943,0.0115,0.0000
C00482=93.306,35.952,48.381,179.9943,0.0115,0.0000
C00483=94.909,31.296,48.237,179.9656,0.1031,0.0000
C00484=95.700,26.654,48.020,-179.9656,1.9485,0.0000
C00485=94.802,22.392,47.807,-178.6053,3.2342,0.0000
C00486=92.454,19.281,47.546,-175.1367,3.7173,0.0000
C00487=89.056,17.687,47.055,-174.3430,2.2287,0.0000
C00488=85.339,16.414,46.074,-176.8237,1.1305,0.0000
C00489=82.045,15.189,44.816,178.2636,-0.7394,0.0000
C00490=79.628,13.762,43.611,169.0403,-7.6243,0.0000
C00491=78.336,11.532,42.745,168.4371,-32.9581,0.0000
C00492=78.220,7.694,42.402,-178.6795,-38.6410,0.0000
C00493=78.467,3.833,42.387,-177.5424,-38.8630,0.0000
C00494=78.562,0.000,42.397,180.0000,-38.8871,0.0000
C00495=78.467,-3.833,42.387,177.5424,-38.8630,0.0000
C00496=78.220,-7.694,42.402,178.6870,-38.6374,0.0000
C00497=78.336,-11.532,42.745,-168.4371,-32.9581,0.0000
C00498=79.628,-13.762,43.611,-169.0403,-7.6243,0.0000
C00499=82.045,-15.189,44.816,-178.2636,-0.7394,0.0000
C00500=85.339,-16.414,46.074,176.8237,1.1305,0.0000
C00501=89.056,-17.687,47.055,174.3430,2.2287,0.0000
C00502=92.454,-19.281,47.546,175.1367,3.7173,0.0000
C00503=94.802,-22.392,47.807,178.6053,3.2342,0.0000
C00504=95.700,-26.654,48.020,179.9656,1.9485,0.0000
C00505=94.909,-31.296,48.237,-179.9656,0.1031,0.0000
C00506=93.306,-35.952,48.381,-179.9943,0.0115,0.0000
C00507=91.399,-40.555,48.381,-179.9943,0.0115,0.0000
C00508=89.240,-44.981,48.237,-179.9484,0.0974,0.0000
C00509=86.517,-48.823,48.020,-178.5957,1.3527,0.0000
C00510=82.869,-51.201,47.807,-176.7315,1.3029,0.0000
C00511=79.009,-51.741,47.546,-173.9433,-0.8124,0.0000
C00512=75.478,-50.465,47.055,-174.4286,-2.4358,0.0000
C00513=71.950,-48.737,46.074,-176.9553,-1.4460,0.0000
C00514=68.755,-47.275,44.816,178.2521,0.7051,0.0000
C00515=66.037,-46.575,43.611,166.9624,2.4236,0.0000
C00516=63.546,-47.238,42.745,148.9091,-17.4211,0.0000
C00517=60.750,-49.870,42.402,151.2284,-30.1838,0.0000
C00518=58.195,-52.774,42.387,151.6554,-30.9681,0.0000
C00519=55.552,-55.552,42.397,150.3051,-29.6949,0.0000
C00520=52.774,-58.195,42.387,149.0319,-28.3446,0.0000
C00521=49.870,-60.750,42.402,149.8193,-28.7685,0.0000
C00522=47.238,-63.546,42.745,162.5789,-31.0909,0.0000
C00523=46.575,-66.037,43.611,-177.5764,-13.0376,0.0000
C00524=47.275,-68.755,44.816,-179.2949,-1.7479,0.0000
C00525=48.737,-71.950,46.074,178.5540,3.0447,0.0000
C00526=50.465,-75.478,47.055,177.5642,5.5714,0.0000
C00527=51.741,-79.009,47.546,179.1876,6.0567,0.0000
C00528=51.201,-82.869,47.807,-178.6971,3.2685,0.0000
C00529=48.823,-86.517,48.020,-178.6473,1.4043,0.0000
C00530=44.981,-89.240,48.237,-179.9026,0.0516,0.0000
C00531=40.555,-91.399,48.381,-179.9885,0.0057,0.0000
C00532=35.952,-93.306,48.381,-179.9885,0.0057,0.0000
C00533=31.296,-94.909,48.237,-179.8969,0.0344,0.0000
C00534=26.654,-95.700,48.020,-178.0515,-0.0344,0.0000
C00535=22.392,-94.802,47.807,-176.7658,-1.3947,0.0000
C00536=19.281,-92.454,47.546,-176.2827,-4.8633,0.0000
C00537=17.687,-89.056,47.055,-177.7713,-5.6570,0.0000
C00538=16.414,-85.339,46.074,-178.8695,-3.1763,0.0000
C00539=15.189,-82.045,44.816,179.2606,1.7364,0.0000
C00540=13.762,-79.628,43.611,172.3757,10.9597,0.0000
C00541=11.532,-78.336,42.745,147.0419,11.5629,0.0000
C00542=7.694,-78.220,42.402,141.3590,-1.3205,0.0000
C00543=3.833,-78.467,42.387,141.1370,-2.4576,0.0000
C00544=0.000,-78.562,42.397,141.1129,0.0000,0.0000
C00545=0.000,-78.562,42.397,141.1129,0.0000,0.0000
C00546=-3.833,-78.467,42.387,141.1370,2.4576,0.0000
C00547=-7.694,-78.220,42.402,141.3626,1.3130,0.0000
C00548=-11.532,-78.336,42.745,147.0419,-11.5629,0.0000
C00549=-13.762,-79.628,43.611,172.3757,-10.9597,0.0000
C00550=-15.189,-82.045,44.816,179.2606,-1.7364,0.0000
C00551=-16.414,-85.339,46.074,-178.8695,3.1763,0.0000
C00552=-17.687,-89.056,47.055,-177.7713,5.6570,0.0000
C00553=-19.281,-92.454,47.546,-176.2827,4.8633,0.0000
C00554=-22.392,-94.802,47.807,-176.7658,1.3947,0.0000
C00555=-26.654,-95.700,48.020,-178.0515,0.0344,0.0000
C00556=-31.296,-94.909,48.237,-179.8969,-0.0344,0.0000
C00557=-35.952,-93.306,48.381,-179.9885,-0.0057,0.0000
C00558=-40.555,-91.399,48.381,-179.9885,-0.0057,0.0000
C00559=-44.981,-89.240,48.237,-179.9026,-0.0516,0.0000
C00560=-48.823,-86.517,48.020,-178.6473,-1.4043,0.0000
C00561=-51.201,-82.869,47.807,-178.6971,-3.2685,0.0000
C00562=-51.741,-79.009,47.546,179.1876,-6.0567,0.0000
C00563=-50.465,-75.478,47.055,177.5642,-5.5714,0.0000
C00564=-48.737,-71.950,46.074,178.5540,-3.0447,0.0000
C00565=-47.275,-68.755,44.816,-179.2949,1.7479,0.0000
C00566=-46.575,-66.037,43.611,-177.5764,13.0376,0.0000
C00567=-47.238,-63.546,42.745,162.5789,31.0909,0.0000
C00568=-49.870,-60.750,42.402,149.8162,28.7716,0.0000
C00569=-52.774,-58.195,42.387,149.0319,28.3446,0.0000
C00570=-55.552,-55.552,42.397,150.3051,29.6949,0.0000
C00571=-58.195,-52.774,42.387,151.6554,30.9681,0.0000
C00572=-60.750,-49.870,42.402,151.2315,30.1807,0.0000
C00573=-63.546,-47.238,42.745,148.9091,17.4211,0.0000
C00574=-66.037,-46.575,43.611,166.9624,-2.4236,0.0000
C00575=-68.755,-47.275,44.816,178.2521,-0.7051,0.0000
C00576=-71.950,-48.737,46.074,-176.9553,1.4460,0.0000
C00577=-75.478,-50.465,47.055,-174.4286,2.4358,0.0000
C00578=-79.009,-51.741,47.546,-173.9433,0.8124,0.0000
C00579=-82.869,-51.201,47.807,-176.7315,-1.3029,0.0000
C00580=-86.517,-48.823,48.020,-178.5957,-1.3527,0.0000
C00581=-89.240,-44.981,48.237,-179.9484,-0.0974,0.0000
C00582=-91.399,-40.555,48.381,-179.9943,-0.0115,0.0000
C00583=-93.306,-35.952,48.381,-179.9943,-0.0115,0.0000
C00584=-94.909,-31.296,48.237,-179.9656,-0.1031,0.0000
C00585=-95.700,-26.654,48.020,179.9656,-1.9485,0.0000
C00586=-94.802,-22.392,47.807,178.6053,-3.2342,0.0000
C00587=-92.454,-19.281,47.546,175.1367,-3.7173,0.0000
C00588=-89.056,-17.687,47.055,174.3430,-2.2287,0.0000
C00589=-85.339,-16.414,46.074,176.8237,-1.1305,0.0000
C00590=-82.045,-15.189,44.816,-178.2636,0.7394,0.0000
C00591=-79.628,-13.762,43.611,-169.0403,7.6243,0.0000
C00592=-78.336,-11.532,42.745,-168.4371,32.9581,0.0000
C00593=-78.220,-7.694,42.402,178.6795,38.6410,0.0000
C00594=-78.467,-3.833,42.387,177.5424,38.8630,0.0000
C00595=-78.562,0.000,42.397,-180.0000,38.8871,0.0000
C00596=-78.467,3.833,42.387,-177.5424,38.8630,0.0000
C00597=-78.220,7.694,42.402,-178.6870,38.6374,0.0000
C00598=-78.336,11.532,42.745,168.4371,32.9581,0.0000
C00599=-79.628,13.762,43.611,169.0403,7.6243,0.0000
C00600=-82.045,15.189,44.816,178.2636,0.7394,0.0000
C00601=-85.339,16.414,46.074,-176.8237,-1.1305,0.0000
C00602=-89.056,17.687,47.055,-174.3430,-2.2287,0.0000
C00603=-92.454,19.281,47.546,-175.1367,-3.7173,0.0000
C00604=-94.802,22.392,47.807,-178.6053,-3.2342,0.0000
C00605=-95.700,26.654,48.020,-179.9656,-1.9485,0.0000
C00606=-94.909,31.296,48.237,179.9656,-0.1031,0.0000
C00607=-93.306,35.952,48.381,179.9943,-0.0115,0.0000
C00608=-91.399,40.555,48.381,179.9943,-0.0115,0.0000
C00609=-89.240,44.981,48.237,179.9484,-0.0974,0.0000
C00610=-86.517,48.823,48.020,178.5957,-1.3527,0.0000
C00611=-82.869,51.201,47.807,176.7315,-1.3029,0.0000
C00612=-79.009,51.741,47.546,173.9433,0.8124,0.0000
C00613=-75.478,50.465,47.055,174.4286,2.4358,0.0000
C00614=-71.950,48.737,46.074,176.9553,1.4460,0.0000
C00615=-68.755,47.275,44.816,-178.2521,-0.7051,0.0000
C00616=-66.037,46.575,43.611,-166.9624,-2.4236,0.0000
C00617=-63.546,47.238,42.745,-148.9091,17.4211,0.0000
C00618=-60.750,49.870,42.402,-151.2284,30.1838,0.0000
C00619=-58.195,52.774,42.387,-151.6554,30.9681,0.0000
C00620=-55.552,55.552,42.397,-150.3051,29.6949,0.0000
C00621=-52.774,58.195,42.387,-149.0319,28.3446,0.0000
C00622=-49.870,60.750,42.402,-149.8193,28.7685,0.0000
C00623=-47.238,63.546,42.745,-162.5789,31.0909,0.0000
C00624=-46.575,66.037,43.611,177.5764,13.0376,0.0000
C00625=-47.275,68.755,44.816,179.2949,1.7479,0.0000
C00626=-48.737,71.950,46.074,-178.5540,-3.0447,0.0000
C00627=-50.465,75.478,47.055,-177.5642,-5.5714,0.0000
C00628=-51.741,79.009,47.546,-179.1876,-6.0567,0.0000
C00629=-51.201,82.869,47.807,178.6971,-3.2685,0.0000
C00630=-48.823,86.517,48.020,178.6473,-1.4043,0.0000
C00631=-44.981,89.240,48.237,179.9026,-0.0516,0.0000
C00632=-40.555,91.399,48.381,179.9885,-0.0057,0.0000
C00633=-35.952,93.306,48.381,179.9885,-0.0057,0.0000
C00634=-31.296,94.909,48.237,179.8969,-0.0344,0.0000
C00635=-26.654,95.700,48.020,178.0515,0.0344,0.0000
C00636=-22.392,94.802,47.807,176.7658,1.3947,0.0000
C00637=-19.281,92.454,47.546,176.2827,4.8633,0.0000
C00638=-17.687,89.056,47.055,177.7713,5.6570,0.0000
C00639=-16.414,85.339,46.074,178.8695,3.1763,0.0000
C00640=-15.189,82.045,44.816,-179.2606,-1.7364,0.0000
C00641=-13.762,79.628,43.611,-172.3757,-10.9597,0.0000
C00642=-11.532,78.336,42.745,-147.0419,-11.5629,0.0000
C00643=-7.694,78.220,42.402,-141.3626,1.3130,0.0000
C00644=-3.833,78.467,42.387,-141.1370,2.4576,0.0000
C00645=0.000,78.562,42.397,-141.1129,0.0000,0.0000
C00646=0.000,77.178,44.107,-140.9053,0.0000,0.0000
C00647=3.707,77.088,44.096,-140.9328,-2.4572,0.0000
C00648=7.481,76.852,44.112,-141.1746,-1.0149,0.0000
C00649=11.270,77.011,44.481,-147.6312,12.5719,0.0000
C00650=13.439,78.412,45.416,-173.7651,9.9152,0.0000
C00651=14.814,81.004,46.718,-179.6734,0.8308,0.0000
C00652=16.001,84.532,48.079,178.7481,-3.8080,0.0000
C00653=17.239,88.522,49.141,177.7633,-6.2161,0.0000
C00654=18.791,92.187,49.674,176.1698,-5.4518,0.0000
C00655=21.929,94.746,49.957,176.4955,-1.6362,0.0000
C00656=26.285,95.767,50.188,177.9196,-0.0688,0.0000
C00657=31.062,94.986,50.423,179.8854,0.0344,0.0000
C00658=35.872,93.336,50.579,179.9885,0.0057,0.0000
C00659=40.633,91.364,50.579,179.9885,0.0057,0.0000
C00660=45.201,89.129,50.423,179.8969,0.0573,0.0000
C00661=49.131,86.304,50.188,178.5784,1.5190,0.0000
C00662=51.489,82.502,49.957,178.6794,3.6303,0.0000
C00663=51.899,78.473,49.674,-178.8465,6.5528,0.0000
C00664=50.405,74.784,49.141,-177.1761,5.9766,0.0000
C00665=48.459,71.088,48.079,-178.1914,3.5792,0.0000
C00666=46.803,67.754,46.718,179.6390,-0.8194,0.0000
C00667=45.943,64.949,45.416,177.3460,-11.3561,0.0000
C00668=46.486,62.424,44.481,-163.8024,-31.2118,0.0000
C00669=49.053,59.633,44.112,-149.8159,-29.0952,0.0000
C00670=51.888,57.130,44.096,-148.8574,-28.5323,0.0000
C00671=54.573,54.573,44.107,-150.1209,-29.8791,0.0000
C00672=57.130,51.888,44.096,-151.4677,-31.1426,0.0000
C00673=59.633,49.053,44.112,-150.9048,-30.1841,0.0000
C00674=62.424,46.486,44.482,-148.7882,-16.2040,0.0000
C00675=64.949,45.943,45.416,-168.6439,2.6540,0.0000
C00676=67.754,46.803,46.718,-179.1806,0.3610,0.0000
C00677=71.088,48.459,48.079,176.4208,-1.8086,0.0000
C00678=74.784,50.405,49.141,174.0234,-2.8239,0.0000
C00679=78.473,51.899,49.674,173.4472,-1.1535,0.0000
C00680=82.502,51.489,49.957,176.3697,1.3206,0.0000
C00681=86.304,49.131,50.188,178.4810,1.4216,0.0000
C00682=89.129,45.201,50.423,179.9427,0.1031,0.0000
C00683=91.364,40.633,50.579,179.9943,0.0115,0.0000
C00684=93.336,35.872,50.579,179.9943,0.0115,0.0000
C00685=94.986,31.062,50.423,179.9656,0.1146,0.0000
C00686=95.767,26.285,50.188,-179.9312,2.0804,0.0000
C00687=94.746,21.929,49.957,-178.3638,3.5045,0.0000
C00688=92.187,18.791,49.674,-174.5482,3.8302,0.0000
C00689=88.522,17.239,49.141,-173.7839,2.2367,0.0000
C00690=84.532,16.001,48.079,-176.1920,1.2519,0.0000
C00691=81.004,14.814,46.718,179.1692,-0.3266,0.0000
C00692=78.412,13.439,45.416,170.0848,-6.2349,0.0000
C00693=77.011,11.270,44.481,167.4281,-32.3688,0.0000
C00694=76.852,7.481,44.112,-178.9851,-38.8254,0.0000
C00695=77.088,3.707,44.096,-177.5428,-39.0672,0.0000
C00696=77.178,0.000,44.107,180.0000,-39.0947,0.0000
C00697=77.088,-3.707,44.096,177.5428,-39.0672,0.0000
C00698=76.852,-7.481,44.112,178.9851,-38.8254,0.0000
C00699=77.011,-11.270,44.482,-167.4281,-32.3688,0.0000
C00700=78.412,-13.439,45.416,-170.0848,-6.2349,0.0000
C00701=81.004,-14.814,46.718,-179.1692,-0.3266,0.0000
C00702=84.532,-16.001,48.079,176.1920,1.2519,0.0000
C00703=88.522,-17.239,49.141,173.7839,2.2367,0.0000
C00704=92.187,-18.791,49.674,174.5482,3.8302,0.0000
C00705=94.746,-21.929,49.957,178.3638,3.5045,0.0000
C00706=95.767,-26.285,50.188,179.9312,2.0804,0.0000
C00707=94.986,-31.062,50.423,-179.9656,0.1146,0.0000
C00708=93.336,-35.872,50.579,-179.9943,0.0115,0.0000
C00709=91.364,-40.633,50.579,-179.9943,0.0115,0.0000
C00710=89.129,-45.201,50.423,-179.9427,0.1031,0.0000
C00711=86.304,-49.131,50.188,-178.4810,1.4216,0.0000
C00712=82.502,-51.489,49.957,-176.3697,1.3206,0.0000
C00713=78.473,-51.899,49.674,-173.4472,-1.1535,0.0000
C00714=74.784,-50.405,49.141,-174.0234,-2.8239,0.0000
C00715=71.088,-48.459,48.079,-176.4208,-1.8086,0.0000
C00716=67.754,-46.803,46.718,179.1806,0.3610,0.0000
C00717=64.949,-45.943,45.416,168.6439,2.6540,0.0000
C00718=62.424,-46.486,44.481,148.7882,-16.1976,0.0000
C00719=59.633,-49.053,44.112,150.9048,-30.1841,0.0000
C00720=57.130,-51.888,44.096,151.4677,-31.1426,0.0000
C00721=54.573,-54.573,44.107,150.1209,-29.8791,0.0000
C00722=51.888,-57.130,44.096,148.8574,-28.5323,0.0000
C00723=49.053,-59.633,44.112,149.8159,-29.0952,0.0000
C00724=46.486,-62.424,44.482,163.7960,-31.2118,0.0000
C00725=45.943,-64.949,45.416,-177.3460,-11.3561,0.0000
C00726=46.803,-67.754,46.718,-179.6390,-0.8194,0.0000
C00727=48.459,-71.088,48.079,178.1914,3.5792,0.0000
C00728=50.405,-74.784,49.141,177.1761,5.9766,0.0000
C00729=51.899,-78.473,49.674,178.8465,6.5528,0.0000
C00730=51.489,-82.502,49.957,-178.6794,3.6303,0.0000
C00731=49.131,-86.304,50.188,-178.5784,1.5190,0.0000
C00732=45.201,-89.129,50.423,-179.8969,0.0573,0.0000
C00733=40.633,-91.364,50.579,-179.9885,0.0057,0.0000
C00734=35.872,-93.336,50.579,-179.9885,0.0057,0.0000
C00735=31.062,-94.986,50.423,-179.8854,0.0344,0.0000
C00736=26.285,-95.767,50.188,-177.9196,-0.0688,0.0000
C00737=21.929,-94.746,49.957,-176.4955,-1.6362,0.0000
C00738=18.791,-92.187,49.674,-176.1698,-5.4518,0.0000
C00739=17.239,-88.522,49.141,-177.7633,-6.2161,0.0000
C00740=16.001,-84.532,48.079,-178.7481,-3.8080,0.0000
C00741=14.814,-81.004,46.718,179.6734,0.8308,0.0000
C00742=13.439,-78.412,45.416,173.7651,9.9152,0.0000
C00743=11.270,-77.011,44.481,147.6312,12.5719,0.0000
C00744=7.481,-76.852,44.112,141.1746,-1.0149,0.0000
C00745=3.707,-77.088,44.096,140.9328,-2.4572,0.0000
C00746=0.000,-77.178,44.107,140.9053,0.0000,0.0000
C00747=0.000,-77.178,44.107,140.9053,0.0000,0.0000
C00748=-3.707,-77.088,44.096,140.9328,2.4572,0.0000
C00749=-7.481,-76.852,44.112,141.1746,1.0149,0.0000
C00750=-11.270,-77.011,44.482,147.6312,-12.5719,0.0000
C00751=-13.439,-78.412,45.416,173.7651,-9.9152,0.0000
C00752=-14.814,-81.004,46.718,179.6734,-0.8308,0.0000
C00753=-16.001,-84.532,48.079,-178.7481,3.8080,0.0000
C00754=-17.239,-88.522,49.141,-177.7633,6.2161,0.0000
C00755=-18.791,-92.187,49.674,-176.1698,5.4518,0.0000
C00756=-21.929,-94.746,49.957,-176.4955,1.6362,0.0000
C00757=-26.285,-95.767,50.188,-177.9196,0.0688,0.0000
C00758=-31.062,-94.986,50.423,-179.8854,-0.0344,0.0000
C00759=-35.872,-93.336,50.579,-179.9885,-0.0057,0.0000
C00760=-40.633,-91.364,50.579,-179.9885,-0.0057,0.0000
C00761=-45.201,-89.129,50.423,-179.8969,-0.0573,0.0000
C00762=-49.131,-86.304,50.188,-178.5784,-1.5190,0.0000
C00763=-51.489,-82.502,49.957,-178.6794,-3.6303,0.0000
C00764=-51.899,-78.473,49.674,178.8465,-6.5528,0.0000
C00765=-50.405,-74.784,49.141,177.1761,-5.9766,0.0000
C00766=-48.459,-71.088,48.079,178.1914,-3.5792,0.0000
C00767=-46.803,-67.754,46.718,-179.6390,0.8194,0.0000
C00768=-45.943,-64.949,45.416,-177.3460,11.3561,0.0000
C00769=-46.486,-62.424,44.481,163.8024,31.2118,0.0000
C00770=-49.053,-59.633,44.112,149.8159,29.0952,0.0000
C00771=-51.888,-57.130,44.096,148.8574,28.5323,0.0000
C00772=-54.573,-54.573,44.107,150.1209,29.8791,0.0000
C00773=-57.130,-51.888,44.096,151.4677,31.1426,0.0000
C00774=-59.633,-49.053,44.112,150.9048,30.1841,0.0000
C00775=-62.424,-46.486,44.482,148.7882,16.2040,0.0000
C00776=-64.949,-45.943,45.416,168.6439,-2.6540,0.0000
C00777=-67.754,-46.803,46.718,179.1806,-0.3610,0.0000
C00778=-71.088,-48.459,48.079,-176.4208,1.8086,0.0000
C00779=-74.784,-50.405,49.141,-174.0234,2.8239,0.0000
C00780=-78.473,-51.899,49.674,-173.4472,1.1535,0.0000
C00781=-82.502,-51.489,49.957,-176.3697,-1.3206,0.0000
C00782=-86.304,-49.131,50.188,-178.4810,-1.4216,0.0000
C00783=-89.129,-45.201,50.423,-179.9427,-0.1031,0.0000
C00784=-91.364,-40.633,50.579,-179.9943,-0.0115,0.0000
C00785=-93.336,-35.872,50.579,-179.9943,-0.0115,0.0000
C00786=-94.986,-31.062,50.423,-179.9656,-0.1146,0.0000
C00787=-95.767,-26.285,50.188,179.9312,-2.0804,0.0000
C00788=-94.746,-21.929,49.957,178.3638,-3.5045,0.0000
C00789=-92.187,-18.791,49.674,174.5482,-3.8302,0.0000
C00790=-88.522,-17.239,49.141,173.7839,-2.2367,0.0000
C00791=-84.532,-16.001,48.079,176.1920,-1.2519,0.0000
C00792=-81.004,-14.814,46.718,-179.1692,0.3266,0.0000
C00793=-78.412,-13.439,45.416,-170.0848,6.2349,0.0000
C00794=-77.011,-11.270,44.481,-167.4281,32.3688,0.0000
C00795=-76.852,-7.481,44.112,178.9851,38.8254,0.0000
C00796=-77.088,-3.707,44.096,177.5428,39.0672,0.0000
C00797=-77.178,0.000,44.107,-180.0000,39.0947,0.0000
C00798=-77.088,3.707,44.096,-177.5428,39.0672,0.0000
C00799=-76.852,7.481,44.112,-178.9851,38.8254,0.0000
C00800=-77.011,11.270,44.482,167.4281,32.3688,0.0000
C00801=-78.412,13.439,45.416,170.0848,6.2349,0.0000
C00802=-81.004,14.814,46.718,179.1692,0.3266,0.0000
C00803=-84.532,16.001,48.079,-176.1920,-1.2519,0.0000
C00804=-88.522,17.239,49.141,-173.7839,-2.2367,0.0000
C00805=-92.187,18.791,49.674,-174.5482,-3.8302,0.0000
C00806=-94.746,21.929,49.957,-178.3638,-3.5045,0.0000
C00807=-95.767,26.285,50.188,-179.9312,-2.0804,0.0000
C00808=-94.986,31.062,50.423,179.9656,-0.1146,0.0000
C00809=-93.336,35.872,50.579,179.9943,-0.0115,0.0000
C00810=-91.364,40.633,50.579,179.9943,-0.0115,0.0000
C00811=-89.129,45.201,50.423,179.9427,-0.1031,0.0000
C00812=-86.304,49.131,50.188,178.4810,-1.4216,0.0000
C00813=-82.502,51.489,49.957,176.3697,-1.3206,0.0000
C00814=-78.473,51.899,49.674,173.4472,1.1535,0.0000
C00815=-74.784,50.405,49.141,174.0234,2.8239,0.0000
C00816=-71.088,48.459,48.079,176.4208,1.8086,0.0000
C00817=-67.754,46.803,46.718,-179.1806,-0.3610,0.0000
C00818=-64.949,45.943,45.416,-168.6439,-2.6540,0.0000
C00819=-62.424,46.486,44.481,-148.7882,16.1976,0.0000
C00820=-59.633,49.053,44.112,-150.9048,30.1841,0.0000
C00821=-57.130,51.888,44.096,-151.4677,31.1426,0.0000
C00822=-54.573,54.573,44.107,-150.1209,29.8791,0.0000
C00823=-51.888,57.130,44.096,-148.8574,28.5323,0.0000
C00824=-49.053,59.633,44.112,-149.8159,29.0952,0.0000
C00825=-46.486,62.424,44.482,-163.7960,31.2118,0.0000
C00826=-45.943,64.949,45.416,177.3460,11.3561,0.0000
C00827=-46.803,67.754,46.718,179.6390,0.8194,0.0000
C00828=-48.459,71.088,48.079,-178.1914,-3.5792,0.0000
C00829=-50.405,74.784,49.141,-177.1761,-5.9766,0.0000
C00830=-51.899,78.473,49.674,-178.8465,-6.5528,0.0000
C00831=-51.489,82.502,49.957,178.6794,-3.6303,0.0000
C00832=-49.131,86.304,50.188,178.5784,-1.5190,0.0000
C00833=-45.201,89.129,50.423,179.8969,-0.0573,0.0000
C00834=-40.633,91.364,50.579,179.9885,-0.0057,0.0000
C00835=-35.872,93.336,50.579,179.9885,-0.0057,0.0000
C00836=-31.062,94.986,50.423,179.8854,-0.0344,0.0000
C00837=-26.285,95.767,50.188,177.9196,0.0688,0.0000
C00838=-21.929,94.746,49.957,176.4955,1.6362,0.0000
C00839=-18.791,92.187,49.674,176.1698,5.4518,0.0000
C00840=-17.239,88.522,49.141,177.7633,6.2161,0.0000
C00841=-16.001,84.532,48.079,178.7481,3.8080,0.0000
C00842=-14.814,81.004,46.718,-179.6734,-0.8308,0.0000
C00843=-13.439,78.412,45.416,-173.7651,-9.9152,0.0000
C00844=-11.270,77.011,44.482,-147.6312,-12.5719,0.0000
C00845=-7.481,76.852,44.112,-141.1746,1.0149,0.0000
C00846=-3.707,77.088,44.096,-140.9328,2.4572,0.0000
C00847=0.000,77.178,44.107,-140.9053,0.0000,0.0000
C00848=0.000,75.789,45.812,-140.7711,0.0000,0.0000
C00849=3.580,75.703,45.801,-140.7985,-2.4398,0.0000
C00850=7.267,75.480,45.818,-141.0646,-0.6998,0.0000
C00851=11.008,75.681,46.215,-148.3523,13.4838,0.0000
C00852=13.116,77.193,47.218,-174.9730,8.8052,0.0000
C00853=14.439,79.961,48.618,-180.0000,0.0057,0.0000
C00854=15.588,83.726,50.084,178.6725,-4.3600,0.0000
C00855=16.791,87.989,51.229,177.7843,-6.6834,0.0000
C00856=18.302,91.921,51.802,176.1258,-5.9660,0.0000
C00857=21.467,94.690,52.107,176.2713,-1.8663,0.0000
C00858=25.919,95.834,52.356,177.8051,-0.1032,0.0000
C00859=30.830,95.062,52.610,179.8739,0.0401,0.0000
C00860=35.794,93.367,52.777,179.9828,0.0057,0.0000
C00861=40.710,91.330,52.777,179.9828,0.0057,0.0000
C00862=45.419,89.019,52.610,179.8854,0.0630,0.0000
C00863=49.437,86.092,52.356,178.5153,1.6222,0.0000
C00864=51.776,82.136,52.107,178.6847,3.9517,0.0000
C00865=52.057,77.939,51.802,-178.5049,6.9409,0.0000
C00866=50.345,74.091,51.229,-176.8224,6.2844,0.0000
C00867=48.181,70.226,50.084,-177.8513,4.0227,0.0000
C00868=46.331,66.751,48.618,180.0000,-0.0057,0.0000
C00869=45.309,63.858,47.218,177.2900,-9.7462,0.0000
C00870=45.731,61.299,46.215,-165.0895,-31.1875,0.0000
C00871=48.234,58.511,45.818,-149.8876,-29.3626,0.0000
C00872=50.999,56.061,45.801,-148.7488,-28.6586,0.0000
C00873=53.591,53.591,45.812,-150.0009,-29.9991,0.0000
C00874=56.061,50.999,45.801,-151.3414,-31.2512,0.0000
C00875=58.511,48.233,45.818,-150.6374,-30.1124,0.0000
C00876=61.299,45.731,46.215,-148.8125,-14.9105,0.0000
C00877=63.858,45.309,47.218,-170.2538,2.7100,0.0000
C00878=66.751,46.331,48.618,-179.9943,0.0000,0.0000
C00879=70.226,48.181,50.084,175.9773,-2.1487,0.0000
C00880=74.091,50.345,51.229,173.7156,-3.1776,0.0000
C00881=77.939,52.057,51.802,173.0591,-1.4951,0.0000
C00882=82.136,51.776,52.107,176.0483,1.3153,0.0000
C00883=86.092,49.437,52.356,178.3778,1.4847,0.0000
C00884=89.019,45.419,52.610,179.9370,0.1146,0.0000
C00885=91.330,40.710,52.777,179.9943,0.0172,0.0000
C00886=93.367,35.794,52.777,179.9943,0.0172,0.0000
C00887=95.062,30.830,52.610,179.9599,0.1261,0.0000
C00888=95.834,25.919,52.356,-179.8968,2.1949,0.0000
C00889=94.690,21.467,52.107,-178.1337,3.7287,0.0000
C00890=91.921,18.302,51.802,-174.0340,3.8742,0.0000
C00891=87.989,16.791,51.229,-173.3166,2.2157,0.0000
C00892=83.726,15.588,50.084,-175.6400,1.3275,0.0000
C00893=79.961,14.439,48.618,179.9943,-0.0000,0.0000
C00894=77.193,13.116,47.218,171.1948,-5.0270,0.0000
C00895=75.681,11.008,46.215,166.5162,-31.6477,0.0000
C00896=75.480,7.267,45.818,-179.3002,-38.9354,0.0000
C00897=75.703,3.580,45.801,-177.5602,-39.2015,0.0000
C00898=75.789,0.000,45.812,180.0000,-39.2289,0.0000
C00899=75.703,-3.580,45.801,177.5602,-39.2015,0.0000
C00900=75.480,-7.267,45.818,179.3002,-38.9354,0.0000
C00901=75.681,-11.008,46.215,-166.5162,-31.6477,0.0000
C00902=77.193,-13.116,47.218,-171.1948,-5.0270,0.0000
C00903=79.961,-14.439,48.618,-179.9943,-0.0000,0.0000
C00904=83.726,-15.588,50.084,175.6400,1.3275,0.0000
C00905=87.989,-16.791,51.229,173.3166,2.2157,0.0000
C00906=91.921,-18.302,51.802,174.0340,3.8742,0.0000
C00907=94.690,-21.467,52.107,178.1337,3.7287,0.0000
C00908=95.834,-25.919,52.356,179.8968,2.1949,0.0000
C00909=95.062,-30.830,52.610,-179.9599,0.1261,0.0000
C00910=93.367,-35.794,52.777,-179.9943,0.0172,0.0000
C00911=91.330,-40.710,52.777,-179.9943,0.0172,0.0000
C00912=89.019,-45.419,52.610,-179.9370,0.1146,0.0000
C00913=86.092,-49.437,52.356,-178.3778,1.4847,0.0000
C00914=82.136,-51.776,52.107,-176.0483,1.3153,0.0000
C00915=77.939,-52.057,51.802,-173.0591,-1.4951,0.0000
C00916=74.091,-50.345,51.229,-173.7156,-3.1776,0.0000
C00917=70.226,-48.181,50.084,-175.9773,-2.1487,0.0000
C00918=66.751,-46.331,48.618,179.9943,0.0000,0.0000
C00919=63.858,-45.309,47.218,170.2538,2.7100,0.0000
C00920=61.299,-45.731,46.215,148.8125,-14.9105,0.0000
C00921=58.511,-48.234,45.818,150.6374,-30.1124,0.0000
C00922=56.061,-50.999,45.801,151.3414,-31.2512,0.0000
C00923=53.591,-53.591,45.812,150.0009,-29.9991,0.0000
C00924=50.999,-56.061,45.801,148.7488,-28.6586,0.0000
C00925=48.233,-58.511,45.818,149.8876,-29.3626,0.0000
C00926=45.731,-61.299,46.215,165.0895,-31.1875,0.0000
C00927=45.309,-63.858,47.218,-177.2900,-9.7462,0.0000
C00928=46.331,-66.751,48.618,-180.0000,-0.0057,0.0000
C00929=48.181,-70.226,50.084,177.8513,4.0227,0.0000
C00930=50.345,-74.091,51.229,176.8224,6.2844,0.0000
C00931=52.057,-77.939,51.802,178.5049,6.9409,0.0000
C00932=51.776,-82.136,52.107,-178.6847,3.9517,0.0000
C00933=49.437,-86.092,52.356,-178.5153,1.6222,0.0000
C00934=45.419,-89.019,52.610,-179.8854,0.0630,0.0000
C00935=40.710,-91.330,52.777,-179.9828,0.0057,0.0000
C00936=35.794,-93.367,52.777,-179.9828,0.0057,0.0000
C00937=30.830,-95.062,52.610,-179.8739,0.0401,0.0000
C00938=25.919,-95.834,52.356,-177.8051,-0.1032,0.0000
C00939=21.467,-94.690,52.107,-176.2713,-1.8663,0.0000
C00940=18.302,-91.921,51.802,-176.1258,-5.9660,0.0000
C00941=16.791,-87.989,51.229,-177.7843,-6.6834,0.0000
C00942=15.588,-83.726,50.084,-178.6725,-4.3600,0.0000
C00943=14.439,-79.961,48.618,180.0000,0.0057,0.0000
C00944=13.116,-77.193,47.218,174.9730,8.8052,0.0000
C00945=11.008,-75.681,46.215,148.3523,13.4838,0.0000
C00946=7.267,-75.480,45.818,141.0646,-0.6998,0.0000
C00947=3.580,-75.703,45.801,140.7985,-2.4398,0.0000
C00948=0.000,-75.789,45.812,140.7711,0.0000,0.0000
C00949=0.000,-75.789,45.812,140.7711,0.0000,0.0000
C00950=-3.580,-75.703,45.801,140.7985,2.4398,0.0000
C00951=-7.267,-75.480,45.818,141.0646,0.6998,0.0000
C00952=-11.008,-75.681,46.215,148.3523,-13.4838,0.0000
C00953=-13.116,-77.193,47.218,174.9730,-8.8052,0.0000
C00954=-14.439,-79.961,48.618,180.0000,-0.0057,0.0000
C00955=-15.588,-83.726,50.084,-178.6725,4.3600,0.0000
C00956=-16.791,-87.989,51.229,-177.7843,6.6834,0.0000
C00957=-18.302,-91.921,51.802,-176.1258,5.9660,0.0000
C00958=-21.467,-94.690,52.107,-176.2713,1.8663,0.0000
C00959=-25.919,-95.834,52.356,-177.8051,0.1032,0.0000
C00960=-30.830,-95.062,52.610,-179.8739,-0.0401,0.0000
C00961=-35.794,-93.367,52.777,-179.9828,-0.0057,0.0000
C00962=-40.710,-91.330,52.777,-179.9828,-0.0057,0.0000
C00963=-45.419,-89.019,52.610,-179.8854,-0.0630,0.0000
C00964=-49.437,-86.092,52.356,-178.5153,-1.6222,0.0000
C00965=-51.776,-82.136,52.107,-178.6847,-3.9517,0.0000
C00966=-52.057,-77.939,51.802,178.5049,-6.9409,0.0000
C00967=-50.345,-74.091,51.229,176.8224,-6.2844,0.0000
C00968=-48.181,-70.226,50.084,177.8513,-4.0227,0.0000
C00969=-46.331,-66.751,48.618,-180.0000,0.0057,0.0000
C00970=-45.309,-63.858,47.218,-177.2900,9.7462,0.0000
C00971=-45.731,-61.299,46.215,165.0895,31.1875,0.0000
C00972=-48.234,-58.511,45.818,149.8876,29.3626,0.0000
C00973=-50.999,-56.061,45.801,148.7488,28.6586,0.0000
C00974=-53.591,-53.591,45.812,150.0009,29.9991,0.0000
C00975=-56.061,-50.999,45.801,151.3414,31.2512,0.0000
C00976=-58.511,-48.233,45.818,150.6374,30.1124,0.0000
C00977=-61.299,-45.731,46.215,148.8125,14.9105,0.0000
C00978=-63.858,-45.309,47.218,170.2538,-2.7100,0.0000
C00979=-66.751,-46.331,48.618,179.9943,-0.0000,0.0000
C00980=-70.226,-48.181,50.084,-175.9773,2.1487,0.0000
C00981=-74.091,-50.345,51.229,-173.7156,3.1776,0.0000
C00982=-77.939,-52.057,51.802,-173.0591,1.4951,0.0000
C00983=-82.136,-51.776,52.107,-176.0483,-1.3153,0.0000
C00984=-86.092,-49.437,52.356,-178.3778,-1.4847,0.0000
C00985=-89.019,-45.419,52.610,-179.9370,-0.1146,0.0000
C00986=-91.330,-40.710,52.777,-179.9943,-0.0172,0.0000
C00987=-93.367,-35.794,52.777,-179.9943,-0.0172,0.0000
C00988=-95.062,-30.830,52.610,-179.9599,-0.1261,0.0000
C00989=-95.834,-25.919,52.356,179.8968,-2.1949,0.0000
C00990=-94.690,-21.467,52.107,178.1337,-3.7287,0.0000
C00991=-91.921,-18.302,51.802,174.0340,-3.8742,0.0000
C00992=-87.989,-16.791,51.229,173.3166,-2.2157,0.0000
C00993=-83.726,-15.588,50.084,175.6400,-1.3275,0.0000
C00994=-79.961,-14.439,48.618,-179.9943,0.0000,0.0000
C00995=-77.193,-13.116,47.218,-171.1948,5.0270,0.0000
C00996=-75.681,-11.008,46.215,-166.5162,31.6477,0.0000
C00997=-75.480,-7.267,45.818,179.3002,38.9354,0.0000
C00998=-75.703,-3.580,45.801,177.5602,39.2015,0.0000
C00999=-75.789,0.000,45.812,-180.0000,39.2289,0.0000
C01000=-75.703,3.580,45.801,-177.5602,39.2015,0.0000
C01001=-75.480,7.267,45.818,-179.3002,38.9354,0.0000
C01002=-75.681,11.008,46.215,166.5162,31.6477,0.0000
C01003=-77.193,13.116,47.218,171.1948,5.0270,0.0000
C01004=-79.961,14.439,48.618,179.9943,0.0000,0.0000
C01005=-83.726,15.588,50.084,-175.6400,-1.3275,0.0000
C01006=-87.989,16.791,51.229,-173.3166,-2.2157,0.0000
C01007=-91.921,18.302,51.802,-174.0340,-3.8742,0.0000
C01008=-94.690,21.467,52.107,-178.1337,-3.7287,0.0000
C01009=-95.834,25.919,52.356,-179.8968,-2.1949,0.0000
C01010=-95.062,30.830,52.610,179.9599,-0.1261,0.0000
C01011=-93.367,35.794,52.777,179.9943,-0.0172,0.0000
C01012=-91.330,40.710,52.777,179.9943,-0.0172,0.0000
C01013=-89.019,45.419,52.610,179.9370,-0.1146,0.0000
C01014=-86.092,49.437,52.356,178.3778,-1.4847,0.0000
C01015=-82.136,51.776,52.107,176.0483,-1.3153,0.0000
C01016=-77.939,52.057,51.802,173.0591,1.4951,0.0000
C01017=-74.091,50.345,51.229,173.7156,3.1776,0.0000
C01018=-70.226,48.181,50.084,175.9773,2.1487,0.0000
C01019=-66.751,46.331,48.618,-179.9943,-0.0000,0.0000
C01020=-63.858,45.309,47.218,-170.2538,-2.7100,0.0000
C01021=-61.299,45.731,46.215,-148.8125,14.9105,0.0000
C01022=-58.511,48.234,45.818,-150.6374,30.1124,0.0000
C01023=-56.061,50.999,45.801,-151.3414,31.2512,0.0000
C01024=-53.591,53.591,45.812,-150.0009,29.9991,0.0000
C01025=-50.999,56.061,45.801,-148.7488,28.6586,0.0000
C01026=-48.233,58.511,45.818,-149.8876,29.3626,0.0000
C01027=-45.731,61.299,46.215,-165.0895,31.1875,0.0000
C01028=-45.309,63.858,47.218,177.2900,9.7462,0.0000
C01029=-46.331,66.751,48.618,180.0000,0.0057,0.0000
C01030=-48.181,70.226,50.084,-177.8513,-4.0227,0.0000
C01031=-50.345,74.091,51.229,-176.8224,-6.2844,0.0000
C01032=-52.057,77.939,51.802,-178.5049,-6.9409,0.0000
C01033=-51.776,82.136,52.107,178.6847,-3.9517,0.0000
C01034=-49.437,86.092,52.356,178.5153,-1.6222,0.0000
C01035=-45.419,89.019,52.610,179.8854,-0.0630,0.0000
C01036=-40.710,91.330,52.777,179.9828,-0.0057,0.0000
C01037=-35.794,93.367,52.777,179.9828,-0.0057,0.0000
C01038=-30.830,95.062,52.610,179.8739,-0.0401,0.0000
C01039=-25.919,95.834,52.356,177.8051,0.1032,0.0000
C01040=-21.467,94.690,52.107,176.2713,1.8663,0.0000
C01041=-18.302,91.921,51.802,176.1258,5.9660,0.0000
C01042=-16.791,87.989,51.229,177.7843,6.6834,0.0000
C01043=-15.588,83.726,50.084,178.6725,4.3600,0.0000
C01044=-14.439,79.961,48.618,-180.0000,-0.0057,0.0000
C01045=-13.116,77.193,47.218,-174.9730,-8.8052,0.0000
C01046=-11.008,75.681,46.215,-148.3523,-13.4838,0.0000
C01047=-7.267,75.480,45.818,-141.0646,0.6998,0.0000
C01048=-3.580,75.703,45.801,-140.7985,2.4398,0.0000
C01049=0.000,75.789,45.812,-140.7711,0.0000,0.0000
C01050=0.000,74.396,47.516,-140.7138,0.0000,0.0000
C01051=3.453,74.315,47.503,-140.7412,-2.4195,0.0000
C01052=7.053,74.105,47.522,-141.0359,-0.3685,0.0000
C01053=10.745,74.349,47.946,-149.2002,14.2818,0.0000
C01054=12.792,75.972,49.019,-176.0136,7.6728,0.0000
C01055=14.064,78.919,50.519,179.7479,-0.7506,0.0000
C01056=15.177,82.922,52.090,178.6314,-4.8312,0.0000
C01057=16.346,87.459,53.317,177.8402,-7.0589,0.0000
C01058=17.816,91.657,53.931,176.1399,-6.3992,0.0000
C01059=21.009,94.635,54.258,176.0982,-2.0852,0.0000
C01060=25.555,95.900,54.525,177.7076,-0.1376,0.0000
C01061=30.600,95.138,54.796,179.8682,0.0401,0.0000
C01062=35.715,93.397,54.976,179.9828,0.0057,0.0000
C01063=40.787,91.296,54.976,179.9828,0.0057,0.0000
C01064=45.636,88.910,54.796,179.8797,0.0630,0.0000
C01065=49.741,85.881,54.525,178.4751,1.7140,0.0000
C01066=52.061,81.773,54.258,178.7129,4.2334,0.0000
C01067=52.213,77.409,53.931,-178.1861,7.2367,0.0000
C01068=50.285,73.401,53.317,-176.5147,6.5177,0.0000
C01069=47.903,69.367,52.090,-177.5456,4.3855,0.0000
C01070=45.859,65.749,50.519,-179.6447,0.7105,0.0000
C01071=44.675,62.766,49.019,177.3651,-8.2299,0.0000
C01072=44.975,60.171,47.946,-166.4258,-31.0310,0.0000
C01073=47.412,57.387,47.522,-150.0381,-29.5676,0.0000
C01074=50.108,54.990,47.503,-148.7075,-28.7229,0.0000
C01075=52.606,52.606,47.516,-149.9539,-30.0461,0.0000
C01076=54.990,50.108,47.503,-151.2771,-31.2925,0.0000
C01077=57.387,47.412,47.522,-150.4324,-29.9619,0.0000
C01078=60.171,44.975,47.946,-148.9690,-13.5807,0.0000
C01079=62.766,44.675,49.019,-171.7701,2.6349,0.0000
C01080=65.749,45.859,50.519,179.2895,-0.3553,0.0000
C01081=69.367,47.903,52.090,175.6145,-2.4544,0.0000
C01082=73.401,50.285,53.317,173.4823,-3.4853,0.0000
C01083=77.409,52.213,53.931,172.7633,-1.8139,0.0000
C01084=81.773,52.061,54.258,175.7666,1.2871,0.0000
C01085=85.881,49.741,54.525,178.2860,1.5249,0.0000
C01086=88.910,45.636,54.796,179.9370,0.1203,0.0000
C01087=91.296,40.787,54.976,179.9943,0.0172,0.0000
C01088=93.397,35.715,54.976,179.9943,0.0172,0.0000
C01089=95.138,30.600,54.796,179.9599,0.1318,0.0000
C01090=95.900,25.555,54.525,-179.8624,2.2924,0.0000
C01091=94.635,21.009,54.258,-177.9148,3.9018,0.0000
C01092=91.657,17.816,53.931,-173.6008,3.8601,0.0000
C01093=87.459,16.346,53.317,-172.9411,2.1598,0.0000
C01094=82.922,15.177,52.090,-175.1688,1.3686,0.0000
C01095=78.919,14.064,50.519,-179.2494,0.2521,0.0000
C01096=75.972,12.792,49.019,172.3272,-3.9864,0.0000
C01097=74.349,10.745,47.946,165.7182,-30.7998,0.0000
C01098=74.105,7.053,47.522,-179.6315,-38.9641,0.0000
C01099=74.315,3.453,47.503,-177.5805,-39.2588,0.0000
C01100=74.396,0.000,47.516,180.0000,-39.2862,0.0000
C01101=74.315,-3.453,47.503,177.5805,-39.2588,0.0000
C01102=74.105,-7.053,47.522,179.6315,-38.9641,0.0000
C01103=74.349,-10.745,47.946,-165.7182,-30.7998,0.0000
C01104=75.972,-12.792,49.019,-172.3272,-3.9864,0.0000
C01105=78.919,-14.064,50.519,179.2494,0.2521,0.0000
C01106=82.922,-15.177,52.090,175.1688,1.3686,0.0000
C01107=87.459,-16.346,53.317,172.9411,2.1598,0.0000
C01108=91.657,-17.816,53.931,173.6008,3.8601,0.0000
C01109=94.635,-21.009,54.258,177.9148,3.9018,0.0000
C01110=95.900,-25.555,54.525,179.8624,2.2924,0.0000
C01111=95.138,-30.600,54.796,-179.9599,0.1318,0.0000
C01112=93.397,-35.715,54.976,-179.9943,0.0172,0.0000
C01113=91.296,-40.787,54.976,-179.9943,0.0172,0.0000
C01114=88.910,-45.636,54.796,-179.9370,0.1203,0.0000
C01115=85.881,-49.741,54.525,-178.2860,1.5249,0.0000
C01116=81.773,-52.061,54.258,-175.7666,1.2871,0.0000
C01117=77.409,-52.213,53.931,-172.7633,-1.8139,0.0000
C01118=73.401,-50.285,53.317,-173.4823,-3.4853,0.0000
C01119=69.367,-47.903,52.090,-175.6145,-2.4544,0.0000
C01120=65.749,-45.859,50.519,-179.2895,-0.3553,0.0000
C01121=62.766,-44.675,49.019,171.7701,2.6349,0.0000
C01122=60.171,-44.975,47.946,148.9690,-13.5742,0.0000
C01123=57.387,-47.412,47.522,150.4324,-29.9619,0.0000
C01124=54.990,-50.108,47.503,151.2771,-31.2925,0.0000
C01125=52.606,-52.606,47.516,149.9539,-30.0461,0.0000
C01126=50.108,-54.990,47.503,148.7075,-28.7229,0.0000
C01127=47.412,-57.387,47.522,150.0381,-29.5676,0.0000
C01128=44.975,-60.171,47.946,166.4193,-31.0310,0.0000
C01129=44.675,-62.766,49.019,-177.3651,-8.2299,0.0000
C01130=45.859,-65.749,50.519,179.6447,0.7105,0.0000
C01131=47.903,-69.367,52.090,177.5456,4.3855,0.0000
C01132=50.285,-73.401,53.317,176.5147,6.5177,0.0000
C01133=52.213,-77.409,53.931,178.1861,7.2367,0.0000
C01134=52.061,-81.773,54.258,-178.7129,4.2334,0.0000
C01135=49.741,-85.881,54.525,-178.4751,1.7140,0.0000
C01136=45.636,-88.910,54.796,-179.8797,0.0630,0.0000
C01137=40.787,-91.296,54.976,-179.9828,0.0057,0.0000
C01138=35.715,-93.397,54.976,-179.9828,0.0057,0.0000
C01139=30.600,-95.138,54.796,-179.8682,0.0401,0.0000
C01140=25.555,-95.900,54.525,-177.7076,-0.1376,0.0000
C01141=21.009,-94.635,54.258,-176.0982,-2.0852,0.0000
C01142=17.816,-91.657,53.931,-176.1399,-6.3992,0.0000
C01143=16.346,-87.459,53.317,-177.8402,-7.0589,0.0000
C01144=15.177,-82.922,52.090,-178.6314,-4.8312,0.0000
C01145=14.064,-78.919,50.519,-179.7479,-0.7506,0.0000
C01146=12.792,-75.972,49.019,176.0136,7.6728,0.0000
C01147=10.745,-74.349,47.946,149.2002,14.2818,0.0000
C01148=7.053,-74.105,47.522,141.0359,-0.3685,0.0000
C01149=3.453,-74.315,47.503,140.7412,-2.4195,0.0000
C01150=0.000,-74.396,47.516,140.7138,0.0000,0.0000
C01151=0.000,-74.396,47.516,140.7138,0.0000,0.0000
C01152=-3.453,-74.315,47.503,140.7412,2.4195,0.0000
C01153=-7.053,-74.105,47.522,141.0359,0.3685,0.0000
C01154=-10.745,-74.349,47.946,149.2002,-14.2818,0.0000
C01155=-12.792,-75.972,49.019,176.0136,-7.6728,0.0000
C01156=-14.064,-78.919,50.519,-179.7479,0.7506,0.0000
C01157=-15.177,-82.922,52.090,-178.6314,4.8312,0.0000
C01158=-16.346,-87.459,53.317,-177.8402,7.0589,0.0000
C01159=-17.816,-91.657,53.931,-176.1399,6.3992,0.0000
C01160=-21.009,-94.635,54.258,-176.0982,2.0852,0.0000
C01161=-25.555,-95.900,54.525,-177.7076,0.1376,0.0000
C01162=-30.600,-95.138,54.796,-179.8682,-0.0401,0.0000
C01163=-35.715,-93.397,54.976,-179.9828,-0.0057,0.0000
C01164=-40.787,-91.296,54.976,-179.9828,-0.0057,0.0000
C01165=-45.636,-88.910,54.796,-179.8797,-0.0630,0.0000
C01166=-49.741,-85.881,54.525,-178.4751,-1.7140,0.0000
C01167=-52.061,-81.773,54.258,-178.7129,-4.2334,0.0000
C01168=-52.213,-77.409,53.931,178.1861,-7.2367,0.0000
C01169=-50.285,-73.401,53.317,176.5147,-6.5177,0.0000
C01170=-47.903,-69.367,52.090,177.5456,-4.3855,0.0000
C01171=-45.859,-65.749,50.519,179.6447,-0.7105,0.0000
C01172=-44.675,-62.766,49.019,-177.3651,8.2299,0.0000
C01173=-44.975,-60.171,47.946,166.4258,31.0310,0.0000
C01174=-47.412,-57.387,47.522,150.0381,29.5676,0.0000
C01175=-50.108,-54.990,47.503,148.7075,28.7229,0.0000
C01176=-52.606,-52.606,47.516,149.9539,30.0461,0.0000
C01177=-54.990,-50.108,47.503,151.2771,31.2925,0.0000
C01178=-57.387,-47.412,47.522,150.4324,29.9619,0.0000
C01179=-60.171,-44.975,47.946,148.9690,13.5807,0.0000
C01180=-62.766,-44.675,49.019,171.7701,-2.6349,0.0000
C01181=-65.749,-45.859,50.519,-179.2895,0.3553,0.0000
C01182=-69.367,-47.903,52.090,-175.6145,2.4544,0.0000
C01183=-73.401,-50.285,53.317,-173.4823,3.4853,0.0000
C01184=-77.409,-52.213,53.931,-172.7633,1.8139,0.0000
C01185=-81.773,-52.061,54.258,-175.7666,-1.2871,0.0000
C01186=-85.881,-49.741,54.525,-178.2860,-1.5249,0.0000
C01187=-88.910,-45.636,54.796,-179.9370,-0.1203,0.0000
C01188=-91.296,-40.787,54.976,-179.9943,-0.0172,0.0000
C01189=-93.397,-35.715,54.976,-179.9943,-0.0172,0.0000
C01190=-95.138,-30.600,54.796,-179.9599,-0.1318,0.0000
C01191=-95.900,-25.555,54.525,179.8624,-2.2924,0.0000
C01192=-94.635,-21.009,54.258,177.9148,-3.9018,0.0000
C01193=-91.657,-17.816,53.931,173.6008,-3.8601,0.0000
C01194=-87.459,-16.346,53.317,172.9411,-2.1598,0.0000
C01195=-82.922,-15.177,52.090,175.1688,-1.3686,0.0000
C01196=-78.919,-14.064,50.519,179.2494,-0.2521,0.0000
C01197=-75.972,-12.792,49.019,-172.3272,3.9864,0.0000
C01198=-74.349,-10.745,47.946,-165.7182,30.7998,0.0000
C01199=-74.105,-7.053,47.522,179.6315,38.9641,0.0000
C01200=-74.315,-3.453,47.503,177.5805,39.2588,0.0000
C01201=-74.396,0.000,47.516,-180.0000,39.2862,0.0000
C01202=-74.315,3.453,47.503,-177.5805,39.2588,0.0000
C01203=-74.105,7.053,47.522,-179.6315,38.9641,0.0000
C01204=-74.349,10.745,47.946,165.7182,30.7998,0.0000
C01205=-75.972,12.792,49.019,172.3272,3.9864,0.0000
C01206=-78.919,14.064,50.519,-179.2494,-0.2521,0.0000
C01207=-82.922,15.177,52.090,-175.1688,-1.3686,0.0000
C01208=-87.459,16.346,53.317,-172.9411,-2.1598,0.0000
C01209=-91.657,17.816,53.931,-173.6008,-3.8601,0.0000
C01210=-94.635,21.009,54.258,-177.9148,-3.9018,0.0000
C01211=-95.900,25.555,54.525,-179.8624,-2.2924,0.0000
C01212=-95.138,30.600,54.796,179.9599,-0.1318,0.0000
C01213=-93.397,35.715,54.976,179.9943,-0.0172,0.0000
C01214=-91.296,40.787,54.976,179.9943,-0.0172,0.0000
C01215=-88.910,45.636,54.796,179.9370,-0.1203,0.0000
C01216=-85.881,49.741,54.525,178.2860,-1.5249,0.0000
C01217=-81.773,52.061,54.258,175.7666,-1.2871,0.0000
C01218=-77.409,52.213,53.931,172.7633,1.8139,0.0000
C01219=-73.401,50.285,53.317,173.4823,3.4853,0.0000
C01220=-69.367,47.903,52.090,175.6145,2.4544,0.0000
C01221=-65.749,45.859,50.519,179.2895,0.3553,0.0000
C01222=-62.766,44.675,49.019,-171.7701,-2.6349,0.0000
C01223=-60.171,44.975,47.946,-148.9690,13.5742,0.0000
C01224=-57.387,47.412,47.522,-150.4324,29.9619,0.0000
C01225=-54.990,50.108,47.503,-151.2771,31.2925,0.0000
C01226=-52.606,52.606,47.516,-149.9539,30.0461,0.0000
C01227=-50.108,54.990,47.503,-148.7075,28.7229,0.0000
C01228=-47.412,57.387,47.522,-150.0381,29.5676,0.0000
C01229=-44.975,60.171,47.946,-166.4193,31.0310,0.0000
C01230=-44.675,62.766,49.019,177.3651,8.2299,0.0000
C01231=-45.859,65.749,50.519,-179.6447,-0.7105,0.0000
C01232=-47.903,69.367,52.090,-177.5456,-4.3855,0.0000
C01233=-50.285,73.401,53.317,-176.5147,-6.5177,0.0000
C01234=-52.213,77.409,53.931,-178.1861,-7.2367,0.0000
C01235=-52.061,81.773,54.258,178.7129,-4.2334,0.0000
C01236=-49.741,85.881,54.525,178.4751,-1.7140,0.0000
C01237=-45.636,88.910,54.796,179.8797,-0.0630,0.0000
C01238=-40.787,91.296,54.976,179.9828,-0.0057,0.0000
C01239=-35.715,93.397,54.976,179.9828,-0.0057,0.0000
C01240=-30.600,95.138,54.796,179.8682,-0.0401,0.0000
C01241=-25.555,95.900,54.525,177.7076,0.1376,0.0000
C01242=-21.009,94.635,54.258,176.0982,2.0852,0.0000
C01243=-17.816,91.657,53.931,176.1399,6.3992,0.0000
C01244=-16.346,87.459,53.317,177.8402,7.0589,0.0000
C01245=-15.177,82.922,52.090,178.6314,4.8312,0.0000
C01246=-14.064,78.919,50.519,179.7479,0.7506,0.0000
C01247=-12.792,75.972,49.019,-176.0136,-7.6728,0.0000
C01248=-10.745,74.349,47.946,-149.2002,-14.2818,0.0000
C01249=-7.053,74.105,47.522,-141.0359,0.3685,0.0000
C01250=-3.453,74.315,47.503,-140.7412,2.4195,0.0000
C01251=0.000,74.396,47.516,-140.7138,0.0000,0.0000
C01252=0.000,73.003,49.219,-140.7299,-0.0000,0.0000
C01253=3.325,72.927,49.205,-140.7574,-2.3967,0.0000
C01254=6.839,72.729,49.225,-141.0807,-0.0221,0.0000
C01255=10.483,73.017,49.677,-150.1610,14.9610,0.0000
C01256=12.469,74.753,50.822,-176.8899,6.5499,0.0000
C01257=13.691,77.880,52.422,179.5587,-1.4268,0.0000
C01258=14.768,82.123,54.099,178.6133,-5.2224,0.0000
C01259=15.905,86.934,55.407,177.9140,-7.3533,0.0000
C01260=17.335,91.395,56.062,176.2009,-6.7511,0.0000
C01261=20.556,94.581,56.410,175.9712,-2.2810,0.0000
C01262=25.196,95.965,56.695,177.6329,-0.1663,0.0000
C01263=30.373,95.213,56.983,179.8625,0.0401,0.0000
C01264=35.638,93.426,57.174,179.9828,0.0057,0.0000
C01265=40.862,91.262,57.174,179.9828,0.0057,0.0000
C01266=45.849,88.802,56.983,179.8739,0.0688,0.0000
C01267=50.042,85.674,56.695,178.4463,1.7944,0.0000
C01268=52.343,81.414,56.410,178.7585,4.4633,0.0000
C01269=52.368,76.884,56.062,-177.8962,7.4401,0.0000
C01270=50.225,72.718,55.407,-176.2535,6.6699,0.0000
C01271=47.627,68.512,54.099,-177.2800,4.6741,0.0000
C01272=45.389,64.750,52.422,-179.3008,1.3237,0.0000
C01273=44.041,61.675,50.822,177.5526,-6.8177,0.0000
C01274=44.219,59.044,49.677,-167.7803,-30.7339,0.0000
C01275=46.591,56.263,49.225,-150.2646,-29.7131,0.0000
C01276=49.216,53.919,49.205,-148.7357,-28.7224,0.0000
C01277=51.621,51.621,49.219,-149.9659,-30.0341,0.0000
C01278=53.919,49.216,49.205,-151.2776,-31.2643,0.0000
C01279=56.263,46.591,49.225,-150.2869,-29.7354,0.0000
C01280=59.044,44.219,49.677,-149.2661,-12.2197,0.0000
C01281=61.675,44.041,50.822,-173.1823,2.4474,0.0000
C01282=64.750,45.389,52.422,178.6763,-0.6992,0.0000
C01283=68.512,47.627,54.099,175.3259,-2.7200,0.0000
C01284=72.718,50.225,55.407,173.3301,-3.7465,0.0000
C01285=76.884,52.368,56.062,172.5599,-2.1038,0.0000
C01286=81.414,52.343,56.410,175.5367,1.2415,0.0000
C01287=85.674,50.042,56.695,178.2056,1.5537,0.0000
C01288=88.802,45.849,56.983,179.9312,0.1261,0.0000
C01289=91.262,40.862,57.174,179.9943,0.0172,0.0000
C01290=93.426,35.638,57.174,179.9943,0.0172,0.0000
C01291=95.213,30.373,56.983,179.9599,0.1375,0.0000
C01292=95.965,25.196,56.695,-179.8337,2.3671,0.0000
C01293=94.581,20.556,56.410,-177.7190,4.0288,0.0000
C01294=91.395,17.335,56.062,-173.2489,3.7991,0.0000
C01295=86.934,15.905,55.407,-172.6467,2.0860,0.0000
C01296=82.123,14.768,54.099,-174.7776,1.3867,0.0000
C01297=77.880,13.691,52.422,-178.5732,0.4413,0.0000
C01298=74.753,12.469,50.822,173.4501,-3.1101,0.0000
C01299=73.017,10.483,49.677,165.0390,-29.8390,0.0000
C01300=72.729,6.839,49.225,-179.9779,-38.9193,0.0000
C01301=72.927,3.325,49.205,-177.6033,-39.2426,0.0000
C01302=73.003,0.000,49.219,-180.0000,-39.2701,0.0000
C01303=72.927,-3.325,49.205,177.6033,-39.2426,0.0000
C01304=72.729,-6.839,49.225,179.9779,-38.9193,0.0000
C01305=73.017,-10.483,49.677,-165.0390,-29.8390,0.0000
C01306=74.753,-12.469,50.822,-173.4501,-3.1101,0.0000
C01307=77.880,-13.691,52.422,178.5732,0.4413,0.0000
C01308=82.123,-14.768,54.099,174.7776,1.3867,0.0000
C01309=86.934,-15.905,55.407,172.6467,2.0860,0.0000
C01310=91.395,-17.335,56.062,173.2489,3.7991,0.0000
C01311=94.581,-20.556,56.410,177.7190,4.0288,0.0000
C01312=95.965,-25.196,56.695,179.8337,2.3671,0.0000
C01313=95.213,-30.373,56.983,-179.9599,0.1375,0.0000
C01314=93.426,-35.638,57.174,-179.9943,0.0172,0.0000
C01315=91.262,-40.862,57.174,-179.9943,0.0172,0.0000
C01316=88.802,-45.849,56.983,-179.9312,0.1261,0.0000
C01317=85.674,-50.042,56.695,-178.2056,1.5537,0.0000
C01318=81.414,-52.343,56.410,-175.5367,1.2415,0.0000
C01319=76.884,-52.368,56.062,-172.5599,-2.1038,0.0000
C01320=72.718,-50.225,55.407,-173.3301,-3.7465,0.0000
C01321=68.512,-47.627,54.099,-175.3259,-2.7200,0.0000
C01322=64.750,-45.389,52.422,-178.6763,-0.6992,0.0000
C01323=61.675,-44.041,50.822,173.1823,2.4474,0.0000
C01324=59.044,-44.219,49.677,149.2661,-12.2197,0.0000
C01325=56.263,-46.591,49.225,150.2869,-29.7354,0.0000
C01326=53.919,-49.216,49.205,151.2776,-31.2643,0.0000
C01327=51.621,-51.621,49.219,149.9659,-30.0341,0.0000
C01328=49.216,-53.919,49.205,148.7357,-28.7224,0.0000
C01329=46.591,-56.263,49.225,150.2646,-29.7131,0.0000
C01330=44.219,-59.044,49.677,167.7803,-30.7339,0.0000
C01331=44.041,-61.675,50.822,-177.5526,-6.8177,0.0000
C01332=45.389,-64.750,52.422,179.3008,1.3237,0.0000
C01333=47.627,-68.512,54.099,177.2800,4.6741,0.0000
C01334=50.225,-72.718,55.407,176.2535,6.6699,0.0000
C01335=52.368,-76.884,56.062,177.8962,7.4401,0.0000
C01336=52.343,-81.414,56.410,-178.7585,4.4633,0.0000
C01337=50.042,-85.674,56.695,-178.4463,1.7944,0.0000
C01338=45.849,-88.802,56.983,-179.8739,0.0688,0.0000
C01339=40.862,-91.262,57.174,-179.9828,0.0057,0.0000
C01340=35.638,-93.426,57.174,-179.9828,0.0057,0.0000
C01341=30.373,-95.213,56.983,-179.8625,0.0401,0.0000
C01342=25.196,-95.965,56.695,-177.6329,-0.1663,0.0000
C01343=20.556,-94.581,56.410,-175.9712,-2.2810,0.0000
C01344=17.335,-91.395,56.062,-176.2009,-6.7511,0.0000
C01345=15.905,-86.934,55.407,-177.9140,-7.3533,0.0000
C01346=14.768,-82.123,54.099,-178.6133,-5.2224,0.0000
C01347=13.691,-77.880,52.422,-179.5587,-1.4268,0.0000
C01348=12.469,-74.753,50.822,176.8899,6.5499,0.0000
C01349=10.483,-73.017,49.677,150.1610,14.9610,0.0000
C01350=6.839,-72.729,49.225,141.0807,-0.0221,0.0000
C01351=3.325,-72.927,49.205,140.7574,-2.3967,0.0000
C01352=0.000,-73.003,49.219,140.7299,-0.0000,0.0000
C01353=0.000,-73.003,49.219,140.7299,-0.0000,0.0000
C01354=-3.325,-72.927,49.205,140.7574,2.3967,0.0000
C01355=-6.839,-72.729,49.225,141.0807,0.0221,0.0000
C01356=-10.483,-73.017,49.677,150.1610,-14.9610,0.0000
C01357=-12.469,-74.753,50.822,176.8899,-6.5499,0.0000
C01358=-13.691,-77.880,52.422,-179.5587,1.4268,0.0000
C01359=-14.768,-82.123,54.099,-178.6133,5.2224,0.0000
C01360=-15.905,-86.934,55.407,-177.9140,7.3533,0.0000
C01361=-17.335,-91.395,56.062,-176.2009,6.7511,0.0000
C01362=-20.556,-94.581,56.410,-175.9712,2.2810,0.0000
C01363=-25.196,-95.965,56.695,-177.6329,0.1663,0.0000
C01364=-30.373,-95.213,56.983,-179.8625,-0.0401,0.0000
C01365=-35.638,-93.426,57.174,-179.9828,-0.0057,0.0000
C01366=-40.862,-91.262,57.174,-179.9828,-0.0057,0.0000
C01367=-45.849,-88.802,56.983,-179.8739,-0.0688,0.0000
C01368=-50.042,-85.674,56.695,-178.4463,-1.7944,0.0000
C01369=-52.343,-81.414,56.410,-178.7585,-4.4633,0.0000
C01370=-52.368,-76.884,56.062,177.8962,-7.4401,0.0000
C01371=-50.225,-72.718,55.407,176.2535,-6.6699,0.0000
C01372=-47.627,-68.512,54.099,177.2800,-4.6741,0.0000
C01373=-45.389,-64.750,52.422,179.3008,-1.3237,0.0000
C01374=-44.041,-61.675,50.822,-177.5526,6.8177,0.0000
C01375=-44.219,-59.044,49.677,167.7803,30.7339,0.0000
C01376=-46.591,-56.263,49.225,150.2646,29.7131,0.0000
C01377=-49.216,-53.919,49.205,148.7357,28.7224,0.0000
C01378=-51.621,-51.621,49.219,149.9659,30.0341,0.0000
C01379=-53.919,-49.216,49.205,151.2776,31.2643,0.0000
C01380=-56.263,-46.591,49.225,150.2869,29.7354,0.0000
C01381=-59.044,-44.219,49.677,149.2661,12.2197,0.0000
C01382=-61.675,-44.041,50.822,173.1823,-2.4474,0.0000
C01383=-64.750,-45.389,52.422,-178.6763,0.6992,0.0000
C01384=-68.512,-47.627,54.099,-175.3259,2.7200,0.0000
C01385=-72.718,-50.225,55.407,-173.3301,3.7465,0.0000
C01386=-76.884,-52.368,56.062,-172.5599,2.1038,0.0000
C01387=-81.414,-52.343,56.410,-175.5367,-1.2415,0.0000
C01388=-85.674,-50.042,56.695,-178.2056,-1.5537,0.0000
C01389=-88.802,-45.849,56.983,-179.9312,-0.1261,0.0000
C01390=-91.262,-40.862,57.174,-179.9943,-0.0172,0.0000
C01391=-93.426,-35.638,57.174,-179.9943,-0.0172,0.0000
C01392=-95.213,-30.373,56.983,-179.9599,-0.1375,0.0000
C01393=-95.965,-25.196,56.695,179.8337,-2.3671,0.0000
C01394=-94.581,-20.556,56.410,177.7190,-4.0288,0.0000
C01395=-91.395,-17.335,56.062,173.2489,-3.7991,0.0000
C01396=-86.934,-15.905,55.407,172.6467,-2.0860,0.0000
C01397=-82.123,-14.768,54.099,174.7776,-1.3867,0.0000
C01398=-77.880,-13.691,52.422,178.5732,-0.4413,0.0000
C01399=-74.753,-12.469,50.822,-173.4501,3.1101,0.0000
C01400=-73.017,-10.483,49.677,-165.0390,29.8390,0.0000
C01401=-72.729,-6.839,49.225,179.9779,38.9193,0.0000
C01402=-72.927,-3.325,49.205,177.6033,39.2426,0.0000
C01403=-73.003,0.000,49.219,180.0000,39.2701,0.0000
C01404=-72.927,3.325,49.205,-177.6033,39.2426,0.0000
C01405=-72.729,6.839,49.225,-179.9779,38.9193,0.0000
C01406=-73.017,10.483,49.677,165.0390,29.8390,0.0000
C01407=-74.753,12.469,50.822,173.4501,3.1101,0.0000
C01408=-77.880,13.691,52.422,-178.5732,-0.4413,0.0000
C01409=-82.123,14.768,54.099,-174.7776,-1.3867,0.0000
C01410=-86.934,15.905,55.407,-172.6467,-2.0860,0.0000
C01411=-91.395,17.335,56.062,-173.2489,-3.7991,0.0000
C01412=-94.581,20.556,56.410,-177.7190,-4.0288,0.0000
C01413=-95.965,25.196,56.695,-179.8337,-2.3671,0.0000
C01414=-95.213,30.373,56.983,179.9599,-0.1375,0.0000
C01415=-93.426,35.638,57.174,179.9943,-0.0172,0.0000
C01416=-91.262,40.862,57.174,179.9943,-0.0172,0.0000
C01417=-88.802,45.849,56.983,179.9312,-0.1261,0.0000
C01418=-85.674,50.042,56.695,178.2056,-1.5537,0.0000
C01419=-81.414,52.343,56.410,175.5367,-1.2415,0.0000
C01420=-76.884,52.368,56.062,172.5599,2.1038,0.0000
C01421=-72.718,50.225,55.407,173.3301,3.7465,0.0000
C01422=-68.512,47.627,54.099,175.3259,2.7200,0.0000
C01423=-64.750,45.389,52.422,178.6763,0.6992,0.0000
C01424=-61.675,44.041,50.822,-173.1823,-2.4474,0.0000
C01425=-59.044,44.219,49.677,-149.2661,12.2197,0.0000
C01426=-56.263,46.591,49.225,-150.2869,29.7354,0.0000
C01427=-53.919,49.216,49.205,-151.2776,31.2643,0.0000
C01428=-51.621,51.621,49.219,-149.9659,30.0341,0.0000
C01429=-49.216,53.919,49.205,-148.7357,28.7224,0.0000
C01430=-46.591,56.263,49.225,-150.2646,29.7131,0.0000
C01431=-44.219,59.044,49.677,-167.7803,30.7339,0.0000
C01432=-44.041,61.675,50.822,177.5526,6.8177,0.0000
C01433=-45.389,64.750,52.422,-179.3008,-1.3237,0.0000
C01434=-47.627,68.512,54.099,-177.2800,-4.6741,0.0000
C01435=-50.225,72.718,55.407,-176.2535,-6.6699,0.0000
C01436=-52.368,76.884,56.062,-177.8962,-7.4401,0.0000
C01437=-52.343,81.414,56.410,178.7585,-4.4633,0.0000
C01438=-50.042,85.674,56.695,178.4463,-1.7944,0.0000
C01439=-45.849,88.802,56.983,179.8739,-0.0688,0.0000
C01440=-40.862,91.262,57.174,179.9828,-0.0057,0.0000
C01441=-35.638,93.426,57.174,179.9828,-0.0057,0.0000
C01442=-30.373,95.213,56.983,179.8625,-0.0401,0.0000
C01443=-25.196,95.965,56.695,177.6329,0.1663,0.0000
C01444=-20.556,94.581,56.410,175.9712,2.2810,0.0000
C01445=-17.335,91.395,56.062,176.2009,6.7511,0.0000
C01446=-15.905,86.934,55.407,177.9140,7.3533,0.0000
C01447=-14.768,82.123,54.099,178.6133,5.2224,0.0000
C01448=-13.691,77.880,52.422,179.5587,1.4268,0.0000
C01449=-12.469,74.753,50.822,-176.8899,-6.5499,0.0000
C01450=-10.483,73.017,49.677,-150.1610,-14.9610,0.0000
C01451=-6.839,72.729,49.225,-141.0807,0.0221,0.0000
C01452=-3.325,72.927,49.205,-140.7574,2.3967,0.0000
C01453=0.000,73.003,49.219,-140.7299,-0.0000,0.0000
C01454=0.000,71.612,50.923,-140.8239,-0.0000,0.0000
C01455=3.198,71.541,50.909,-140.8469,-2.3567,0.0000
C01456=6.625,71.354,50.929,-141.2069,0.3308,0.0000
C01457=10.220,71.688,51.410,-151.2324,15.5127,0.0000
C01458=12.146,73.537,52.627,-177.6280,5.4561,0.0000
C01459=13.319,76.847,54.328,179.4152,-2.0288,0.0000
C01460=14.363,81.331,56.111,178.6183,-5.5452,0.0000
C01461=15.469,86.415,57.500,178.0055,-7.5666,0.0000
C01462=16.861,91.137,58.195,176.2973,-7.0161,0.0000
C01463=20.110,94.527,58.564,175.8846,-2.4536,0.0000
C01464=24.842,96.029,58.865,177.5757,-0.2007,0.0000
C01465=30.149,95.287,59.171,179.8568,0.0458,0.0000
C01466=35.562,93.456,59.373,179.9828,0.0057,0.0000
C01467=40.937,91.230,59.373,179.9828,0.0057,0.0000
C01468=46.059,88.697,59.171,179.8682,0.0688,0.0000
C01469=50.337,85.469,58.865,178.4291,1.8517,0.0000
C01470=52.621,81.060,58.564,178.8215,4.6413,0.0000
C01471=52.521,76.366,58.195,-177.6412,7.5624,0.0000
C01472=50.167,72.043,57.500,-176.0389,6.7582,0.0000
C01473=47.354,67.666,56.111,-177.0428,4.8942,0.0000
C01474=44.921,63.757,54.328,-178.9795,1.8513,0.0000
C01475=43.410,60.587,52.627,177.8120,-5.5303,0.0000
C01476=43.464,57.918,51.410,-169.1332,-30.3054,0.0000
C01477=45.770,55.140,50.929,-150.5592,-29.7908,0.0000
C01478=48.325,52.849,50.909,-148.8334,-28.6627,0.0000
C01479=50.637,50.637,50.923,-150.0478,-29.9522,0.0000
C01480=52.848,48.326,50.909,-151.3373,-31.1666,0.0000
C01481=55.140,45.770,50.930,-150.2092,-29.4352,0.0000
C01482=57.918,43.464,51.410,-149.6946,-10.8668,0.0000
C01483=60.587,43.410,52.627,-174.4697,2.1880,0.0000
C01484=63.757,44.921,54.328,178.1487,-1.0205,0.0000
C01485=67.666,47.354,56.111,175.1058,-2.9572,0.0000
C01486=72.043,50.167,57.500,173.2418,-3.9611,0.0000
C01487=76.366,52.521,58.195,172.4376,-2.3588,0.0000
C01488=81.060,52.621,58.564,175.3587,1.1785,0.0000
C01489=85.469,50.337,58.865,178.1483,1.5709,0.0000
C01490=88.697,46.059,59.171,179.9312,0.1318,0.0000
C01491=91.230,40.937,59.373,179.9943,0.0172,0.0000
C01492=93.456,35.562,59.373,179.9943,0.0172,0.0000
C01493=95.287,30.149,59.171,179.9542,0.1432,0.0000
C01494=96.029,24.842,58.865,-179.7993,2.4243,0.0000
C01495=94.527,20.110,58.564,-177.5464,4.1154,0.0000
C01496=91.137,16.861,58.195,-172.9839,3.7027,0.0000
C01497=86.415,15.469,57.500,-172.4334,1.9945,0.0000
C01498=81.331,14.363,56.111,-174.4548,1.3817,0.0000
C01499=76.847,13.319,54.328,-177.9712,0.5848,0.0000
C01500=73.537,12.146,52.627,174.5439,-2.3720,0.0000
C01501=71.688,10.220,51.410,164.4873,-28.7676,0.0000
C01502=71.354,6.625,50.929,179.6692,-38.7931,0.0000
C01503=71.541,3.198,50.909,-177.6433,-39.1531,0.0000
C01504=71.612,0.000,50.923,-180.0000,-39.1761,0.0000
C01505=71.541,-3.198,50.909,177.6433,-39.1531,0.0000
C01506=71.354,-6.626,50.930,-179.6692,-38.7931,0.0000
C01507=71.688,-10.221,51.410,-164.4873,-28.7676,0.0000
C01508=73.537,-12.146,52.627,-174.5439,-2.3720,0.0000
C01509=76.847,-13.319,54.328,177.9712,0.5848,0.0000
C01510=81.331,-14.363,56.111,174.4548,1.3817,0.0000
C01511=86.415,-15.469,57.500,172.4334,1.9945,0.0000
C01512=91.137,-16.861,58.195,172.9839,3.7027,0.0000
C01513=94.527,-20.110,58.564,177.5464,4.1154,0.0000
C01514=96.029,-24.842,58.865,179.7993,2.4243,0.0000
C01515=95.287,-30.149,59.171,-179.9542,0.1432,0.0000
C01516=93.456,-35.562,59.373,-179.9943,0.0172,0.0000
C01517=91.230,-40.937,59.373,-179.9943,0.0172,0.0000
C01518=88.697,-46.059,59.171,-179.9312,0.1318,0.0000
C01519=85.469,-50.337,58.865,-178.1483,1.5709,0.0000
C01520=81.060,-52.621,58.564,-175.3587,1.1785,0.0000
C01521=76.366,-52.521,58.195,-172.4376,-2.3588,0.0000
C01522=72.043,-50.167,57.500,-173.2418,-3.9611,0.0000
C01523=67.666,-47.354,56.111,-175.1058,-2.9572,0.0000
C01524=63.757,-44.921,54.328,-178.1487,-1.0205,0.0000
C01525=60.587,-43.410,52.627,174.4697,2.1880,0.0000
C01526=57.918,-43.464,51.410,149.6946,-10.8668,0.0000
C01527=55.140,-45.770,50.929,150.2092,-29.4408,0.0000
C01528=52.849,-48.325,50.909,151.3373,-31.1666,0.0000
C01529=50.637,-50.637,50.923,150.0478,-29.9522,0.0000
C01530=48.326,-52.848,50.909,148.8334,-28.6627,0.0000
C01531=45.770,-55.140,50.930,150.5648,-29.7908,0.0000
C01532=43.464,-57.918,51.410,169.1332,-30.3054,0.0000
C01533=43.410,-60.587,52.627,-177.8120,-5.5303,0.0000
C01534=44.921,-63.757,54.328,178.9795,1.8513,0.0000
C01535=47.354,-67.666,56.111,177.0428,4.8942,0.0000
C01536=50.167,-72.043,57.500,176.0389,6.7582,0.0000
C01537=52.521,-76.366,58.195,177.6412,7.5624,0.0000
C01538=52.621,-81.060,58.564,-178.8215,4.6413,0.0000
C01539=50.337,-85.469,58.865,-178.4291,1.8517,0.0000
C01540=46.059,-88.697,59.171,-179.8682,0.0688,0.0000
C01541=40.937,-91.230,59.373,-179.9828,0.0057,0.0000
C01542=35.562,-93.456,59.373,-179.9828,0.0057,0.0000
C01543=30.149,-95.287,59.171,-179.8568,0.0458,0.0000
C01544=24.842,-96.029,58.865,-177.5757,-0.2007,0.0000
C01545=20.110,-94.527,58.564,-175.8846,-2.4536,0.0000
C01546=16.861,-91.137,58.195,-176.2973,-7.0161,0.0000
C01547=15.469,-86.415,57.500,-178.0055,-7.5666,0.0000
C01548=14.363,-81.331,56.111,-178.6183,-5.5452,0.0000
C01549=13.319,-76.847,54.328,-179.4152,-2.0288,0.0000
C01550=12.146,-73.537,52.627,177.6280,5.4561,0.0000
C01551=10.220,-71.688,51.410,151.2324,15.5127,0.0000
C01552=6.625,-71.354,50.929,141.2069,0.3308,0.0000
C01553=3.198,-71.541,50.909,140.8469,-2.3567,0.0000
C01554=0.000,-71.612,50.923,140.8239,-0.0000,0.0000
C01555=0.000,-71.612,50.923,140.8239,-0.0000,0.0000
C01556=-3.198,-71.541,50.909,140.8469,2.3567,0.0000
C01557=-6.626,-71.354,50.930,141.2069,-0.3308,0.0000
C01558=-10.221,-71.688,51.410,151.2324,-15.5127,0.0000
C01559=-12.146,-73.537,52.627,177.6280,-5.4561,0.0000
C01560=-13.319,-76.847,54.328,-179.4152,2.0288,0.0000
C01561=-14.363,-81.331,56.111,-178.6183,5.5452,0.0000
C01562=-15.469,-86.415,57.500,-178.0055,7.5666,0.0000
C01563=-16.861,-91.137,58.195,-176.2973,7.0161,0.0000
C01564=-20.110,-94.527,58.564,-175.8846,2.4536,0.0000
C01565=-24.842,-96.029,58.865,-177.5757,0.2007,0.0000
C01566=-30.149,-95.287,59.171,-179.8568,-0.0458,0.0000
C01567=-35.562,-93.456,59.373,-179.9828,-0.0057,0.0000
C01568=-40.937,-91.230,59.373,-179.9828,-0.0057,0.0000
C01569=-46.059,-88.697,59.171,-179.8682,-0.0688,0.0000
C01570=-50.337,-85.469,58.865,-178.4291,-1.8517,0.0000
C01571=-52.621,-81.060,58.564,-178.8215,-4.6413,0.0000
C01572=-52.521,-76.366,58.195,177.6412,-7.5624,0.0000
C01573=-50.167,-72.043,57.500,176.0389,-6.7582,0.0000
C01574=-47.354,-67.666,56.111,177.0428,-4.8942,0.0000
C01575=-44.921,-63.757,54.328,178.9795,-1.8513,0.0000
C01576=-43.410,-60.587,52.627,-177.8120,5.5303,0.0000
C01577=-43.464,-57.918,51.410,169.1332,30.3054,0.0000
C01578=-45.770,-55.140,50.929,150.5592,29.7908,0.0000
C01579=-48.325,-52.849,50.909,148.8334,28.6627,0.0000
C01580=-50.637,-50.637,50.923,150.0478,29.9522,0.0000
C01581=-52.848,-48.326,50.909,151.3373,31.1666,0.0000
C01582=-55.140,-45.770,50.930,150.2092,29.4352,0.0000
C01583=-57.918,-43.464,51.410,149.6946,10.8668,0.0000
C01584=-60.587,-43.410,52.627,174.4697,-2.1880,0.0000
C01585=-63.757,-44.921,54.328,-178.1487,1.0205,0.0000
C01586=-67.666,-47.354,56.111,-175.1058,2.9572,0.0000
C01587=-72.043,-50.167,57.500,-173.2418,3.9611,0.0000
C01588=-76.366,-52.521,58.195,-172.4376,2.3588,0.0000
C01589=-81.060,-52.621,58.564,-175.3587,-1.1785,0.0000
C01590=-85.469,-50.337,58.865,-178.1483,-1.5709,0.0000
C01591=-88.697,-46.059,59.171,-179.9312,-0.1318,0.0000
C01592=-91.230,-40.937,59.373,-179.9943,-0.0172,0.0000
C01593=-93.456,-35.562,59.373,-179.9943,-0.0172,0.0000
C01594=-95.287,-30.149,59.171,-179.9542,-0.1432,0.0000
C01595=-96.029,-24.842,58.865,179.7993,-2.4243,0.0000
C01596=-94.527,-20.110,58.564,177.5464,-4.1154,0.0000
C01597=-91.137,-16.861,58.195,172.9839,-3.7027,0.0000
C01598=-86.415,-15.469,57.500,172.4334,-1.9945,0.0000
C01599=-81.331,-14.363,56.111,174.4548,-1.3817,0.0000
C01600=-76.847,-13.319,54.328,177.9712,-0.5848,0.0000
C01601=-73.537,-12.146,52.627,-174.5439,2.3720,0.0000
C01602=-71.688,-10.220,51.410,-164.4873,28.7676,0.0000
C01603=-71.354,-6.625,50.929,-179.6692,38.7931,0.0000
C01604=-71.541,-3.198,50.909,177.6433,39.1531,0.0000
C01605=-71.612,0.000,50.923,180.0000,39.1761,0.0000
C01606=-71.541,3.198,50.909,-177.6433,39.1531,0.0000
C01607=-71.354,6.626,50.930,179.6692,38.7931,0.0000
C01608=-71.688,10.221,51.410,164.4873,28.7676,0.0000
C01609=-73.537,12.146,52.627,174.5439,2.3720,0.0000
C01610=-76.847,13.319,54.328,-177.9712,-0.5848,0.0000
C01611=-81.331,14.363,56.111,-174.4548,-1.3817,0.0000
C01612=-86.415,15.469,57.500,-172.4334,-1.9945,0.0000
C01613=-91.137,16.861,58.195,-172.9839,-3.7027,0.0000
C01614=-94.527,20.110,58.564,-177.5464,-4.1154,0.0000
C01615=-96.029,24.842,58.865,-179.7993,-2.4243,0.0000
C01616=-95.287,30.149,59.171,179.9542,-0.1432,0.0000
C01617=-93.456,35.562,59.373,179.9943,-0.0172,0.0000
C01618=-91.230,40.937,59.373,179.9943,-0.0172,0.0000
C01619=-88.697,46.059,59.171,179.9312,-0.1318,0.0000
C01620=-85.469,50.337,58.865,178.1483,-1.5709,0.0000
C01621=-81.060,52.621,58.564,175.3587,-1.1785,0.0000
C01622=-76.366,52.521,58.195,172.4376,2.3588,0.0000
C01623=-72.043,50.167,57.500,173.2418,3.9611,0.0000
C01624=-67.666,47.354,56.111,175.1058,2.9572,0.0000
C01625=-63.757,44.921,54.328,178.1487,1.0205,0.0000
C01626=-60.587,43.410,52.627,-174.4697,-2.1880,0.0000
C01627=-57.918,43.464,51.410,-149.6946,10.8668,0.0000
C01628=-55.140,45.770,50.929,-150.2092,29.4408,0.0000
C01629=-52.849,48.325,50.909,-151.3373,31.1666,0.0000
C01630=-50.637,50.637,50.923,-150.0478,29.9522,0.0000
C01631=-48.326,52.848,50.909,-148.8334,28.6627,0.0000
C01632=-45.770,55.140,50.930,-150.5648,29.7908,0.0000
C01633=-43.464,57.918,51.410,-169.1332,30.3054,0.0000
C01634=-43.410,60.587,52.627,177.8120,5.5303,0.0000
C01635=-44.921,63.757,54.328,-178.9795,-1.8513,0.0000
C01636=-47.354,67.666,56.111,-177.0428,-4.8942,0.0000
C01637=-50.167,72.043,57.500,-176.0389,-6.7582,0.0000
C01638=-52.521,76.366,58.195,-177.6412,-7.5624,0.0000
C01639=-52.621,81.060,58.564,178.8215,-4.6413,0.0000
C01640=-50.337,85.469,58.865,178.4291,-1.8517,0.0000
C01641=-46.059,88.697,59.171,179.8682,-0.0688,0.0000
C01642=-40.937,91.230,59.373,179.9828,-0.0057,0.0000
C01643=-35.562,93.456,59.373,179.9828,-0.0057,0.0000
C01644=-30.149,95.287,59.171,179.8568,-0.0458,0.0000
C01645=-24.842,96.029,58.865,177.5757,0.2007,0.0000
C01646=-20.110,94.527,58.564,175.8846,2.4536,0.0000
C01647=-16.861,91.137,58.195,176.2973,7.0161,0.0000
C01648=-15.469,86.415,57.500,178.0055,7.5666,0.0000
C01649=-14.363,81.331,56.111,178.6183,5.5452,0.0000
C01650=-13.319,76.847,54.328,179.4152,2.0288,0.0000
C01651=-12.146,73.537,52.627,-177.6280,-5.4561,0.0000
C01652=-10.221,71.688,51.410,-151.2324,-15.5127,0.0000
C01653=-6.626,71.354,50.930,-141.2069,-0.3308,0.0000
C01654=-3.198,71.541,50.909,-140.8469,2.3567,0.0000
C01655=0.000,71.612,50.923,-140.8239,-0.0000,0.0000
C01656=0.000,70.224,52.630,-140.9867,-0.0000,0.0000
C01657=3.072,70.158,52.615,-141.0099,-2.3145,0.0000
C01658=6.412,69.984,52.637,-141.4109,0.6890,0.0000
C01659=9.959,70.362,53.146,-152.4014,15.9357,0.0000
C01660=11.825,72.328,54.436,-178.2356,4.4066,0.0000
C01661=12.951,75.822,56.240,179.3117,-2.5565,0.0000
C01662=13.963,80.549,58.128,178.6407,-5.7927,0.0000
C01663=15.041,85.905,59.597,178.1034,-7.6988,0.0000
C01664=16.396,90.884,60.330,176.4229,-7.1948,0.0000
C01665=19.672,94.474,60.719,175.8441,-2.5973,0.0000
C01666=24.496,96.092,61.037,177.5470,-0.2294,0.0000
C01667=29.931,95.359,61.359,179.8510,0.0458,0.0000
C01668=35.488,93.484,61.571,179.9828,0.0057,0.0000
C01669=41.009,91.197,61.571,179.9828,0.0057,0.0000
C01670=46.265,88.593,61.359,179.8625,0.0745,0.0000
C01671=50.626,85.269,61.037,178.4233,1.8975,0.0000
C01672=52.893,80.714,60.719,178.8961,4.7674,0.0000
C01673=52.671,75.858,60.330,-177.4211,7.6045,0.0000
C01674=50.109,71.379,59.597,-175.8712,6.7880,0.0000
C01675=47.084,66.830,58.128,-176.8521,5.0562,0.0000
C01676=44.457,62.772,56.240,-178.6810,2.2931,0.0000
C01677=42.782,59.505,54.436,178.1265,-4.3609,0.0000
C01678=42.712,56.796,53.146,-170.4717,-29.7492,0.0000
C01679=44.952,54.020,52.637,-150.9354,-29.8041,0.0000
C01680=47.437,51.781,52.615,-148.9950,-28.5386,0.0000
C01681=49.656,49.656,52.630,-150.1885,-29.8060,0.0000
C01682=51.781,47.437,52.615,-151.4614,-31.0050,0.0000
C01683=54.020,44.952,52.637,-150.1959,-29.0646,0.0000
C01684=56.796,42.711,53.146,-150.2508,-9.5283,0.0000
C01685=59.505,42.782,54.436,-175.6391,1.8735,0.0000
C01686=62.772,44.457,56.240,177.7069,-1.3190,0.0000
C01687=66.830,47.084,58.128,174.9438,-3.1479,0.0000
C01688=71.379,50.109,59.597,173.2120,-4.1288,0.0000
C01689=75.858,52.671,60.330,172.3955,-2.5789,0.0000
C01690=80.714,52.893,60.719,175.2326,1.1039,0.0000
C01691=85.269,50.626,61.037,178.1025,1.5767,0.0000
C01692=88.593,46.265,61.359,179.9255,0.1375,0.0000
C01693=91.197,41.009,61.571,179.9943,0.0172,0.0000
C01694=93.484,35.488,61.571,179.9943,0.0172,0.0000
C01695=95.359,29.931,61.359,179.9542,0.1490,0.0000
C01696=96.092,24.496,61.037,-179.7706,2.4530,0.0000
C01697=94.474,19.672,60.719,-177.4027,4.1559,0.0000
C01698=90.884,16.396,60.330,-172.8052,3.5771,0.0000
C01699=85.905,15.041,59.597,-172.3012,1.8966,0.0000
C01700=80.549,13.963,58.128,-174.2073,1.3593,0.0000
C01701=75.822,12.951,56.240,-177.4435,0.6883,0.0000
C01702=72.328,11.825,54.436,175.5934,-1.7644,0.0000
C01703=70.362,9.959,53.146,164.0643,-27.5986,0.0000
C01704=69.984,6.412,52.637,179.3110,-38.5891,0.0000
C01705=70.158,3.072,52.615,-177.6855,-38.9901,0.0000
C01706=70.224,0.000,52.630,-180.0000,-39.0133,0.0000
C01707=70.158,-3.071,52.615,177.6855,-38.9901,0.0000
C01708=69.984,-6.412,52.637,-179.3110,-38.5891,0.0000
C01709=70.362,-9.959,53.146,-164.0705,-27.6038,0.0000
C01710=72.328,-11.825,54.436,-175.5934,-1.7644,0.0000
C01711=75.822,-12.951,56.240,177.4435,0.6883,0.0000
C01712=80.549,-13.963,58.128,174.2073,1.3593,0.0000
C01713=85.905,-15.041,59.597,172.3012,1.8966,0.0000
C01714=90.884,-16.396,60.330,172.8052,3.5771,0.0000
C01715=94.474,-19.672,60.719,177.4027,4.1559,0.0000
C01716=96.092,-24.496,61.037,179.7706,2.4530,0.0000
C01717=95.359,-29.931,61.359,-179.9542,0.1490,0.0000
C01718=93.484,-35.488,61.571,-179.9943,0.0172,0.0000
C01719=91.197,-41.009,61.571,-179.9943,0.0172,0.0000
C01720=88.593,-46.265,61.359,-179.9255,0.1375,0.0000
C01721=85.269,-50.626,61.037,-178.1025,1.5767,0.0000
C01722=80.714,-52.893,60.719,-175.2326,1.1039,0.0000
C01723=75.858,-52.671,60.330,-172.3955,-2.5789,0.0000
C01724=71.379,-50.109,59.597,-173.2120,-4.1288,0.0000
C01725=66.830,-47.084,58.128,-174.9438,-3.1479,0.0000
C01726=62.772,-44.457,56.240,-177.7069,-1.3190,0.0000
C01727=59.505,-42.782,54.436,175.6391,1.8735,0.0000
C01728=56.796,-42.712,53.146,150.2508,-9.5283,0.0000
C01729=54.020,-44.952,52.637,150.1959,-29.0646,0.0000
C01730=51.781,-47.437,52.615,151.4614,-31.0050,0.0000
C01731=49.656,-49.656,52.630,150.1940,-29.8115,0.0000
C01732=47.437,-51.781,52.615,148.9950,-28.5386,0.0000
C01733=44.952,-54.020,52.637,150.9354,-29.8041,0.0000
C01734=42.711,-56.796,53.146,170.4717,-29.7492,0.0000
C01735=42.782,-59.505,54.436,-178.1265,-4.3609,0.0000
C01736=44.457,-62.772,56.240,178.6810,2.2931,0.0000
C01737=47.084,-66.830,58.128,176.8521,5.0562,0.0000
C01738=50.109,-71.379,59.597,175.8712,6.7880,0.0000
C01739=52.671,-75.858,60.330,177.4211,7.6045,0.0000
C01740=52.893,-80.714,60.719,-178.8961,4.7674,0.0000
C01741=50.626,-85.269,61.037,-178.4233,1.8975,0.0000
C01742=46.265,-88.593,61.359,-179.8625,0.0745,0.0000
C01743=41.009,-91.197,61.571,-179.9828,0.0057,0.0000
C01744=35.488,-93.484,61.571,-179.9828,0.0057,0.0000
C01745=29.931,-95.359,61.359,-179.8510,0.0458,0.0000
C01746=24.496,-96.092,61.037,-177.5470,-0.2294,0.0000
C01747=19.672,-94.474,60.719,-175.8441,-2.5973,0.0000
C01748=16.396,-90.884,60.330,-176.4229,-7.1948,0.0000
C01749=15.041,-85.905,59.597,-178.1034,-7.6988,0.0000
C01750=13.963,-80.549,58.128,-178.6407,-5.7927,0.0000
C01751=12.951,-75.822,56.240,-179.3117,-2.5565,0.0000
C01752=11.825,-72.328,54.436,178.2356,4.4066,0.0000
C01753=9.959,-70.362,53.146,152.4014,15.9357,0.0000
C01754=6.412,-69.984,52.637,141.4109,0.6890,0.0000
C01755=3.072,-70.158,52.615,141.0099,-2.3145,0.0000
C01756=0.000,-70.224,52.630,140.9867,-0.0000,0.0000
C01757=0.000,-70.224,52.630,140.9867,-0.0000,0.0000
C01758=-3.071,-70.158,52.615,141.0099,2.3145,0.0000
C01759=-6.412,-69.984,52.637,141.4109,-0.6890,0.0000
C01760=-9.959,-70.362,53.146,152.3962,-15.9295,0.0000
C01761=-11.825,-72.328,54.436,178.2356,-4.4066,0.0000
C01762=-12.951,-75.822,56.240,-179.3117,2.5565,0.0000
C01763=-13.963,-80.549,58.128,-178.6407,5.7927,0.0000
C01764=-15.041,-85.905,59.597,-178.1034,7.6988,0.0000
C01765=-16.396,-90.884,60.330,-176.4229,7.1948,0.0000
C01766=-19.672,-94.474,60.719,-175.8441,2.5973,0.0000
C01767=-24.496,-96.092,61.037,-177.5470,0.2294,0.0000
C01768=-29.931,-95.359,61.359,-179.8510,-0.0458,0.0000
C01769=-35.488,-93.484,61.571,-179.9828,-0.0057,0.0000
C01770=-41.009,-91.197,61.571,-179.9828,-0.0057,0.0000
C01771=-46.265,-88.593,61.359,-179.8625,-0.0745,0.0000
C01772=-50.626,-85.269,61.037,-178.4233,-1.8975,0.0000
C01773=-52.893,-80.714,60.719,-178.8961,-4.7674,0.0000
C01774=-52.671,-75.858,60.330,177.4211,-7.6045,0.0000
C01775=-50.109,-71.379,59.597,175.8712,-6.7880,0.0000
C01776=-47.084,-66.830,58.128,176.8521,-5.0562,0.0000
C01777=-44.457,-62.772,56.240,178.6810,-2.2931,0.0000
C01778=-42.782,-59.505,54.436,-178.1265,4.3609,0.0000
C01779=-42.712,-56.796,53.146,170.4717,29.7492,0.0000
C01780=-44.952,-54.020,52.637,150.9354,29.8041,0.0000
C01781=-47.437,-51.781,52.615,148.9950,28.5386,0.0000
C01782=-49.656,-49.656,52.630,150.1885,29.8060,0.0000
C01783=-51.781,-47.437,52.615,151.4614,31.0050,0.0000
C01784=-54.020,-44.952,52.637,150.1959,29.0646,0.0000
C01785=-56.796,-42.711,53.146,150.2508,9.5283,0.0000
C01786=-59.505,-42.782,54.436,175.6391,-1.8735,0.0000
C01787=-62.772,-44.457,56.240,-177.7069,1.3190,0.0000
C01788=-66.830,-47.084,58.128,-174.9438,3.1479,0.0000
C01789=-71.379,-50.109,59.597,-173.2120,4.1288,0.0000
C01790=-75.858,-52.671,60.330,-172.3955,2.5789,0.0000
C01791=-80.714,-52.893,60.719,-175.2326,-1.1039,0.0000
C01792=-85.269,-50.626,61.037,-178.1025,-1.5767,0.0000
C01793=-88.593,-46.265,61.359,-179.9255,-0.1375,0.0000
C01794=-91.197,-41.009,61.571,-179.9943,-0.0172,0.0000
C01795=-93.484,-35.488,61.571,-179.9943,-0.0172,0.0000
C01796=-95.359,-29.931,61.359,-179.9542,-0.1490,0.0000
C01797=-96.092,-24.496,61.037,179.7706,-2.4530,0.0000
C01798=-94.474,-19.672,60.719,177.4027,-4.1559,0.0000
C01799=-90.884,-16.396,60.330,172.8052,-3.5771,0.0000
C01800=-85.905,-15.041,59.597,172.3012,-1.8966,0.0000
C01801=-80.549,-13.963,58.128,174.2073,-1.3593,0.0000
C01802=-75.822,-12.951,56.240,177.4435,-0.6883,0.0000
C01803=-72.328,-11.825,54.436,-175.5934,1.7644,0.0000
C01804=-70.362,-9.959,53.146,-164.0643,27.5986,0.0000
C01805=-69.984,-6.412,52.637,-179.3110,38.5891,0.0000
C01806=-70.158,-3.072,52.615,177.6855,38.9901,0.0000
C01807=-70.224,0.000,52.630,180.0000,39.0133,0.0000
C01808=-70.158,3.071,52.615,-177.6855,38.9901,0.0000
C01809=-69.984,6.412,52.637,179.3110,38.5891,0.0000
C01810=-70.362,9.959,53.146,164.0705,27.6038,0.0000
C01811=-72.328,11.825,54.436,175.5934,1.7644,0.0000
C01812=-75.822,12.951,56.240,-177.4435,-0.6883,0.0000
C01813=-80.549,13.963,58.128,-174.2073,-1.3593,0.0000
C01814=-85.905,15.041,59.597,-172.3012,-1.8966,0.0000
C01815=-90.884,16.396,60.330,-172.8052,-3.5771,0.0000
C01816=-94.474,19.672,60.719,-177.4027,-4.1559,0.0000
C01817=-96.092,24.496,61.037,-179.7706,-2.4530,0.0000
C01818=-95.359,29.931,61.359,179.9542,-0.1490,0.0000
C01819=-93.484,35.488,61.571,179.9943,-0.0172,0.0000
C01820=-91.197,41.009,61.571,179.9943,-0.0172,0.0000
C01821=-88.593,46.265,61.359,179.9255,-0.1375,0.0000
C01822=-85.269,50.626,61.037,178.1025,-1.5767,0.0000
C01823=-80.714,52.893,60.719,175.2326,-1.1039,0.0000
C01824=-75.858,52.671,60.330,172.3955,2.5789,0.0000
C01825=-71.379,50.109,59.597,173.2120,4.1288,0.0000
C01826=-66.830,47.084,58.128,174.9438,3.1479,0.0000
C01827=-62.772,44.457,56.240,177.7069,1.3190,0.0000
C01828=-59.505,42.782,54.436,-175.6391,-1.8735,0.0000
C01829=-56.796,42.712,53.146,-150.2508,9.5283,0.0000
C01830=-54.020,44.952,52.637,-150.1959,29.0646,0.0000
C01831=-51.781,47.437,52.615,-151.4614,31.0050,0.0000
C01832=-49.656,49.656,52.630,-150.1940,29.8115,0.0000
C01833=-47.437,51.781,52.615,-148.9950,28.5386,0.0000
C01834=-44.952,54.020,52.637,-150.9354,29.8041,0.0000
C01835=-42.711,56.796,53.146,-170.4717,29.7492,0.0000
C01836=-42.782,59.505,54.436,178.1265,4.3609,0.0000
C01837=-44.457,62.772,56.240,-178.6810,-2.2931,0.0000
C01838=-47.084,66.830,58.128,-176.8521,-5.0562,0.0000
C01839=-50.109,71.379,59.597,-175.8712,-6.7880,0.0000
C01840=-52.671,75.858,60.330,-177.4211,-7.6045,0.0000
C01841=-52.893,80.714,60.719,178.8961,-4.7674,0.0000
C01842=-50.626,85.269,61.037,178.4233,-1.8975,0.0000
C01843=-46.265,88.593,61.359,179.8625,-0.0745,0.0000
C01844=-41.009,91.197,61.571,179.9828,-0.0057,0.0000
C01845=-35.488,93.484,61.571,179.9828,-0.0057,0.0000
C01846=-29.931,95.359,61.359,179.8510,-0.0458,0.0000
C01847=-24.496,96.092,61.037,177.5470,0.2294,0.0000
C01848=-19.672,94.474,60.719,175.8441,2.5973,0.0000
C01849=-16.396,90.884,60.330,176.4229,7.1948,0.0000
C01850=-15.041,85.905,59.597,178.1034,7.6988,0.0000
C01851=-13.963,80.549,58.128,178.6407,5.7927,0.0000
C01852=-12.951,75.822,56.240,179.3117,2.5565,0.0000
C01853=-11.825,72.328,54.436,-178.2356,-4.4066,0.0000
C01854=-9.959,70.362,53.146,-152.3962,-15.9295,0.0000
C01855=-6.412,69.984,52.637,-141.4109,-0.6890,0.0000
C01856=-3.071,70.158,52.615,-141.0099,2.3145,0.0000
C01857=0.000,70.224,52.630,-140.9867,-0.0000,0.0000
C01858=0.000,68.843,54.342,-141.2230,-0.0000,0.0000
C01859=2.945,68.781,54.326,-141.2462,-2.2627,0.0000
C01860=6.200,68.619,54.350,-141.6928,1.0514,0.0000
C01861=9.699,69.044,54.888,-153.6494,16.2173,0.0000
C01862=11.507,71.127,56.252,-178.7372,3.4233,0.0000
C01863=12.586,74.809,58.158,179.2369,-3.0041,0.0000
C01864=13.569,79.780,60.151,178.6806,-5.9712,0.0000
C01865=14.621,85.405,61.698,178.2072,-7.7564,0.0000
C01866=15.942,90.636,62.469,176.5671,-7.2973,0.0000
C01867=19.246,94.423,62.877,175.8494,-2.7066,0.0000
C01868=24.159,96.154,63.210,177.5356,-0.2523,0.0000
C01869=29.718,95.429,63.547,179.8510,0.0458,0.0000
C01870=35.416,93.512,63.770,179.9828,0.0057,0.0000
C01871=41.080,91.166,63.770,179.9828,0.0057,0.0000
C01872=46.465,88.493,63.547,179.8625,0.0745,0.0000
C01873=50.908,85.074,63.210,178.4348,1.9204,0.0000
C01874=53.158,80.376,62.877,178.9707,4.8422,0.0000
